(* IEC 61131-3 sources: elnaProjects/ElpcLogic/PomarKc7Unchanged/build_USO_ecl (part 5) *)

  resetDiProtection(protections.OsevojSdvigPravyjDi);
  resetDiProtection(protections.OsevojSdvigLevyjDi);
  resetDiProtection(protections.dP_masloGaz_LowDI);
  resetDiProtection(protections.DavlenieMaslaSmazkiDi);
  resetDiProtection(protections.mvOff);
  resetDiProtection(protections.NeispravnostVozbuzhdenijaDi);
  resetDiProtection(protections.AO_KC);
  resetDiProtection(protections.AO_PRU);
  resetDiProtection(protections.AO_SHU);
  resetDiProtection(protections.Srab_BEAO);
  resetDiProtection(protections.EAO_PRU);
  resetDiProtection(protections.BEAO_knSHU);
  resetDiProtection(protections.Kran1sdvig);
  resetDiProtection(protections.Kran2sdvig);
END_FUNCTION

FUNCTION BlockAllIM : BOOL
  VAR_IN_OUT
    IM : ImConfig;
  END_VAR

  IF NOT IM.Kran1.inOpcCommandsDisabled   THEN IM.Kran1.inOpcCommandsDisabled:=TRUE; END_IF;
  IF NOT IM.Kran2.inOpcCommandsDisabled   THEN IM.Kran2.inOpcCommandsDisabled:=TRUE; END_IF;
  IF NOT IM.Kran3b.inOpcCommandsDisabled  THEN IM.Kran3b.inOpcCommandsDisabled:=TRUE; END_IF;
  IF NOT IM.Kran4.inOpcCommandsDisabled   THEN IM.Kran4.inOpcCommandsDisabled:=TRUE; END_IF;
  IF NOT IM.Kran5.inOpcCommandsDisabled   THEN IM.Kran5.inOpcCommandsDisabled:=TRUE; END_IF;
  (*IF NOT IM.Kran6.inOpcCommandsDisabled   THEN IM.Kran6.inOpcCommandsDisabled:=TRUE; END_IF;*)

  IF NOT IM.nu1.inOpcCommandsDisabled     THEN IM.nu1.inOpcCommandsDisabled:=TRUE; END_IF;
  IF NOT IM.nu2.inOpcCommandsDisabled     THEN IM.nu2.inOpcCommandsDisabled:=TRUE; END_IF;
  IF NOT IM.pns.inOpcCommandsDisabled     THEN IM.pns.inOpcCommandsDisabled:=TRUE; END_IF;
  IF NOT IM.v1_Avom.inOpcCommandsDisabled THEN IM.v1_Avom.inOpcCommandsDisabled:=TRUE; END_IF;
  IF NOT IM.v2_Avom.inOpcCommandsDisabled THEN IM.v2_Avom.inOpcCommandsDisabled:=TRUE; END_IF;
  IF NOT IM.Ten.inOpcCommandsDisabled     THEN IM.Ten.inOpcCommandsDisabled:=TRUE; END_IF;
  IF NOT IM.mv.inOpcCommandsDisabled      THEN IM.mv.inOpcCommandsDisabled:=TRUE; END_IF;
END_FUNCTION

FUNCTION UnBlockAllIM : BOOL
  VAR_IN_OUT
    IM : ImConfig;
  END_VAR

  IF IM.TypeSwitch.Value = 1 THEN

  IF IM.Kran1.inOpcCommandsDisabled   THEN IM.Kran1.inOpcCommandsDisabled:=FALSE; END_IF;
  IF IM.Kran2.inOpcCommandsDisabled   THEN IM.Kran2.inOpcCommandsDisabled:=FALSE; END_IF;
  IF IM.Kran3b.inOpcCommandsDisabled  THEN IM.Kran3b.inOpcCommandsDisabled:=FALSE; END_IF;
  IF IM.Kran4.inOpcCommandsDisabled   THEN IM.Kran4.inOpcCommandsDisabled:=FALSE; END_IF;
  IF IM.Kran5.inOpcCommandsDisabled   THEN IM.Kran5.inOpcCommandsDisabled:=FALSE; END_IF;
  (*IF IM.Kran6.inOpcCommandsDisabled   THEN IM.Kran6.inOpcCommandsDisabled:=FALSE; END_IF;*)
  END_IF;

  IF IM.nu1.inOpcCommandsDisabled     THEN IM.nu1.inOpcCommandsDisabled:=FALSE; END_IF;
  IF IM.nu2.inOpcCommandsDisabled     THEN IM.nu2.inOpcCommandsDisabled:=FALSE; END_IF;
  IF IM.pns.inOpcCommandsDisabled     THEN IM.pns.inOpcCommandsDisabled:=FALSE; END_IF;
  IF IM.v1_Avom.inOpcCommandsDisabled THEN IM.v1_Avom.inOpcCommandsDisabled:=FALSE; END_IF;
  IF IM.v2_Avom.inOpcCommandsDisabled THEN IM.v2_Avom.inOpcCommandsDisabled:=FALSE; END_IF;
  IF IM.Ten.inOpcCommandsDisabled     THEN IM.Ten.inOpcCommandsDisabled:=FALSE; END_IF;
  IF IM.mv.inOpcCommandsDisabled      THEN IM.mv.inOpcCommandsDisabled:=FALSE; END_IF;
END_FUNCTION

FUNCTION_BLOCK RemontAlg
  VAR_IN_OUT
    StrAlg : struct_Alg;
  END_VAR
  VAR
    _sunpackerCommand : fb_sunpackerCommand;
    source : BYTE;
    cmd : BYTE;
    lastCmd : BYTE;
    source_for_Status : BYTE;
    cmd_for_Status : BYTE;
    command_error_for_Status : BYTE;
    resetCmdTimer : TON;
    resetCmdTimerPriznak : BOOL;
  END_VAR
  VAR_EXTERNAL
    protectManager : struct_ProtectionsManager;
    algManager : struct_AlgoritmsManager;
    ModeGpa : TYPE_ModeGpa;
    PMcommand : TYPE_CommandsPotectionsManager;
    IM : ImConfig;
  END_VAR

  StrAlg.CanRun := StrAlg.inCanRun;
  StrAlg.OpcCommandsDisabled := StrAlg.inOpcCommandsDisabled;

  (* ---- Если управление с ВУ заблокировано, то передаем команду из алгоритма ---- *)
  IF StrAlg.inOpcCommandsDisabled THEN
  	StrAlg.inCommand := StrAlg.inCommand_Alg;
  ELSE (* иначе передаем команду с АРМа*)
  	StrAlg.inCommand := StrAlg.inCommand_ARM;
  END_IF;

  _sunpackerCommand(command := StrAlg.inCommand);
  	source := _sunpackerCommand.source;
  	cmd := _sunpackerCommand.cmd;

  IF cmd <> 0 AND lastCmd <> cmd AND (((NOT StrAlg.opcCommandsDisabled) AND source > 0) OR source = 0) then
  	CASE BYTE_TO_INT(cmd) OF
  		(*cmdRun*) 1: 	IF (StrAlg.CanRun) THEN
  					StrAlg.isRuning := TRUE;
  					StrAlg.isEnded := FALSE;
  					StrAlg.hasError 	:= FALSE;
                                               (*****************       OnRun       *****************)
                                                        algManager.nMode:=ModeGpa.MODE_REMONT;
                                                        protectManager.inCommand:=PMcommand.ResetAllProtections;
  					    UnBlockAllIM(IM);
                                                    (*StrAlg.inOpcCommandsDisabled:=FALSE;*)
  					cmd_for_Status := cmd;
  					source_for_Status := source;
  					command_error_for_Status := 0;
  				ELSE
  					StrAlg.isRuning := FALSE;
  					StrAlg.isEnded := FALSE;
  					StrAlg.hasError 	:= FALSE;

  					cmd_for_Status := 0;
  					source_for_Status := source;
  					command_error_for_Status := cmd;
  				END_IF;
  		(*cmdReset*) 2: 	StrAlg.isRuning := FALSE;
  				StrAlg.isEnded := FALSE;
  				StrAlg.hasError 	:= FALSE;
                                          (*****************       OnReset       *****************)
                                                    BlockAllIM(IM);
                                                    protectManager.inCommand:=PMcommand.RestartAllProtections;
                                                    algManager.nMode:=ModeGpa.MODE_STOP;

  				cmd_for_Status := cmd;
  				source_for_Status := source;
  				command_error_for_Status := 0;
  	END_CASE;
  	resetCmdTimer(IN := false);
  	resetCmdTimerPriznak := TRUE;
  END_IF;
  lastCmd := cmd;

  resetCmdTimer(IN := resetCmdTimerPriznak, PT := T#5S);
  IF resetCmdTimer.Q THEN
  	resetCmdTimerPriznak := FALSE;
  	source_for_Status := 0;
  	cmd_for_Status := 0;
  	command_error_for_Status := 0;
  END_IF;

  StrAlg.status :=  SHL(BYTE_TO_DWORD(source_for_Status), 29)
  			OR SHL(BYTE_TO_DWORD(cmd_for_Status), 26)
  			OR SHL(BYTE_TO_DWORD(command_error_for_Status), 23)
  			OR SHL(BOOL_TO_DWORD(StrAlg.OpcCommandsDisabled ), 21)
  			OR SHL(BOOL_TO_DWORD(StrAlg.hasError),4)
  			OR SHL(BOOL_TO_DWORD(StrAlg.CanRun),2)
  			OR SHL(BOOL_TO_DWORD(StrAlg.isEnded),1)
  			OR BOOL_TO_DWORD(StrAlg.isRuning);
END_FUNCTION_BLOCK

FUNCTION EnableAiLimits : BOOL
  VAR_IN_OUT
    ai : AiConfig;
  END_VAR

  ai.P_masla_smazki_nizkoe.Disabled_LA:=FALSE;
   ai.P_masla_smazki_nizkoe.Disabled_LW:=FALSE;
   ai.P_masla_smazki_srednee_posle_nasosov.Disabled_LW:=FALSE;
   ai.dPmaslo_gaz.Disabled_LA:=FALSE;
   ai.dPmaslo_gaz.Disabled_LW:=FALSE;
END_FUNCTION

FUNCTION DisableAiLimits : BOOL
  VAR_IN_OUT
    ai : AiConfig;
  END_VAR

  ai.P_masla_smazki_nizkoe.Disabled_LA:=TRUE;
   ai.P_masla_smazki_nizkoe.Disabled_LW:=TRUE;
   ai.P_masla_smazki_srednee_posle_nasosov.Disabled_LW:=TRUE;
   ai.dPmaslo_gaz.Disabled_LA:=TRUE;
   ai.dPmaslo_gaz.Disabled_LW:=TRUE;
END_FUNCTION

FUNCTION_BLOCK TestProtectionAlg
  VAR_IN_OUT
    StrAlg : struct_Alg;
  END_VAR
  VAR
    _sunpackerCommand : fb_sunpackerCommand;
    source : BYTE;
    cmd : BYTE;
    lastCmd : BYTE;
    source_for_Status : BYTE;
    cmd_for_Status : BYTE;
    command_error_for_Status : BYTE;
    resetCmdTimer : TON;
    resetCmdTimerPriznak : BOOL;
  END_VAR
  VAR_EXTERNAL
    ai : AiConfig;
    protectManager : struct_ProtectionsManager;
    algManager : struct_AlgoritmsManager;
    ModeGpa : TYPE_ModeGpa;
    PMcommand : TYPE_CommandsPotectionsManager;
    IM : ImConfig;
  END_VAR

  StrAlg.CanRun := StrAlg.inCanRun;
  StrAlg.OpcCommandsDisabled := StrAlg.inOpcCommandsDisabled;

  (* ---- Если управление с ВУ заблокировано, то передаем команду из алгоритма ---- *)
  IF StrAlg.inOpcCommandsDisabled THEN
  	StrAlg.inCommand := StrAlg.inCommand_Alg;
  ELSE (* иначе передаем команду с АРМа*)
  	StrAlg.inCommand := StrAlg.inCommand_ARM;
  END_IF;

  _sunpackerCommand(command := StrAlg.inCommand);
  	source := _sunpackerCommand.source;
  	cmd := _sunpackerCommand.cmd;

  IF cmd <> 0 AND lastCmd <> cmd AND (((NOT StrAlg.opcCommandsDisabled) AND source > 0) OR source = 0) then
  	CASE BYTE_TO_INT(cmd) OF
  		(*cmdRun*) 1: 	IF (StrAlg.CanRun) THEN
  					StrAlg.isRuning := TRUE;
  					StrAlg.isEnded := FALSE;
  					StrAlg.hasError 	:= FALSE;
                                               (*****************       OnRun       *****************)
                                                        algManager.nMode:=ModeGpa.MODE_TESTAZ;
                                                        protectManager.inCommand:=PMcommand.CheckProtections;
  					    EnableAiLimits(ai);
                                                        IM.SingleSignals.P_oil_low.Disabled_Sig:=FALSE;
                                                        IM.SingleSignals.dP_oilgaz_low.Disabled_Sig:=FALSE;
                                                    (*StrAlg.inOpcCommandsDisabled:=FALSE;*)
  					cmd_for_Status := cmd;
  					source_for_Status := source;
  					command_error_for_Status := 0;
  				ELSE
  					StrAlg.isRuning := FALSE;
  					StrAlg.isEnded := FALSE;
  					StrAlg.hasError 	:= FALSE;

  					cmd_for_Status := 0;
  					source_for_Status := source;
  					command_error_for_Status := cmd;
  				END_IF;
  		(*cmdReset*) 2: 	StrAlg.isRuning := FALSE;
  				StrAlg.isEnded := FALSE;
  				StrAlg.hasError 	:= FALSE;
                                          (*****************       OnReset       *****************)
                                                    DisableAiLimits(ai);
                                                    IM.SingleSignals.P_oil_low.Disabled_Sig:=TRUE;
                                                    IM.SingleSignals.dP_oilgaz_low.Disabled_Sig:=TRUE;
                                                    protectManager.inCommand:=PMcommand.RestartAllProtections;
                                                    algManager.nMode:=ModeGpa.MODE_STOP;

  				cmd_for_Status := cmd;
  				source_for_Status := source;
  				command_error_for_Status := 0;
  	END_CASE;
  	resetCmdTimer(IN := false);
  	resetCmdTimerPriznak := TRUE;
  END_IF;
  lastCmd := cmd;

  resetCmdTimer(IN := resetCmdTimerPriznak, PT := T#5S);
  IF resetCmdTimer.Q THEN
  	resetCmdTimerPriznak := FALSE;
  	source_for_Status := 0;
  	cmd_for_Status := 0;
  	command_error_for_Status := 0;
  END_IF;

  StrAlg.status :=  SHL(BYTE_TO_DWORD(source_for_Status), 29)
  			OR SHL(BYTE_TO_DWORD(cmd_for_Status), 26)
  			OR SHL(BYTE_TO_DWORD(command_error_for_Status), 23)
  			OR SHL(BOOL_TO_DWORD(StrAlg.OpcCommandsDisabled ), 21)
  			OR SHL(BOOL_TO_DWORD(StrAlg.hasError),4)
  			OR SHL(BOOL_TO_DWORD(StrAlg.CanRun),2)
  			OR SHL(BOOL_TO_DWORD(StrAlg.isEnded),1)
  			OR BOOL_TO_DWORD(StrAlg.isRuning);
END_FUNCTION_BLOCK

FUNCTION_BLOCK TestImAlg
  VAR_IN_OUT
    StrAlg : struct_Alg;
  END_VAR
  VAR
    _sunpackerCommand : fb_sunpackerCommand;
    source : BYTE;
    cmd : BYTE;
    lastCmd : BYTE;
    source_for_Status : BYTE;
    cmd_for_Status : BYTE;
    command_error_for_Status : BYTE;
    resetCmdTimer : TON;
    resetCmdTimerPriznak : BOOL;
  END_VAR
  VAR_EXTERNAL
    protectManager : struct_ProtectionsManager;
    algManager : struct_AlgoritmsManager;
    ModeGpa : TYPE_ModeGpa;
    PMcommand : TYPE_CommandsPotectionsManager;
    IM : ImConfig;
  END_VAR

  StrAlg.CanRun := StrAlg.inCanRun;
  StrAlg.OpcCommandsDisabled := StrAlg.inOpcCommandsDisabled;

  (* ---- Если управление с ВУ заблокировано, то передаем команду из алгоритма ---- *)
  IF StrAlg.inOpcCommandsDisabled THEN
  	StrAlg.inCommand := StrAlg.inCommand_Alg;
  ELSE (* иначе передаем команду с АРМа*)
  	StrAlg.inCommand := StrAlg.inCommand_ARM;
  END_IF;

  _sunpackerCommand(command := StrAlg.inCommand);
  	source := _sunpackerCommand.source;
  	cmd := _sunpackerCommand.cmd;

  IF cmd <> 0 AND lastCmd <> cmd AND (((NOT StrAlg.opcCommandsDisabled) AND source > 0) OR source = 0) then
  	CASE BYTE_TO_INT(cmd) OF
  		(*cmdRun*) 1: 	IF (StrAlg.CanRun) THEN
  					StrAlg.isRuning := TRUE;
  					StrAlg.isEnded := FALSE;
  					StrAlg.hasError 	:= FALSE;
                                               (*****************       OnRun       *****************)

                                                        algManager.nMode:=ModeGpa.MODE_TESTIM;
  					    UnBlockAllIM(IM);

                                                    (*StrAlg.inOpcCommandsDisabled:=FALSE;*)
  					cmd_for_Status := cmd;
  					source_for_Status := source;
  					command_error_for_Status := 0;
  				ELSE
  					StrAlg.isRuning := FALSE;
  					StrAlg.isEnded := FALSE;
  					StrAlg.hasError 	:= FALSE;

  					cmd_for_Status := 0;
  					source_for_Status := source;
  					command_error_for_Status := cmd;
  				END_IF;
  		(*cmdReset*) 2: 	StrAlg.isRuning := FALSE;
  				StrAlg.isEnded := FALSE;
  				StrAlg.hasError 	:= FALSE;
                                          (*****************       OnReset       *****************)
                                                    BlockAllIM(IM);
                                                    algManager.nMode:=ModeGpa.MODE_STOP;

  				cmd_for_Status := cmd;
  				source_for_Status := source;
  				command_error_for_Status := 0;
  	END_CASE;
  	resetCmdTimer(IN := false);
  	resetCmdTimerPriznak := TRUE;
  END_IF;
  lastCmd := cmd;

  resetCmdTimer(IN := resetCmdTimerPriznak, PT := T#5S);
  IF resetCmdTimer.Q THEN
  	resetCmdTimerPriznak := FALSE;
  	source_for_Status := 0;
  	cmd_for_Status := 0;
  	command_error_for_Status := 0;
  END_IF;

  StrAlg.status :=  SHL(BYTE_TO_DWORD(source_for_Status), 29)
  			OR SHL(BYTE_TO_DWORD(cmd_for_Status), 26)
  			OR SHL(BYTE_TO_DWORD(command_error_for_Status), 23)
  			OR SHL(BOOL_TO_DWORD(StrAlg.OpcCommandsDisabled ), 21)
  			OR SHL(BOOL_TO_DWORD(StrAlg.hasError),4)
  			OR SHL(BOOL_TO_DWORD(StrAlg.CanRun),2)
  			OR SHL(BOOL_TO_DWORD(StrAlg.isEnded),1)
  			OR BOOL_TO_DWORD(StrAlg.isRuning);
END_FUNCTION_BLOCK

FUNCTION_BLOCK fb_AutoTenAlg
  VAR_IN_OUT
    StrAlg : struct_Alg;
    PNS : struct_Switch;
    TEN : struct_Switch;
  END_VAR
  VAR_INPUT
    T_masla : struct_AI;
    Uroven_masla : struct_AI;
    offTemperature : struct_AnalogParametr;
  END_VAR
  VAR
    _sunpackerCommand : fb_sunpackerCommand;
    _statusAi : TYPE_StatusAi;
    _statusDualInput : TYPE_statusDualInput;
    _commandDualInput : TYPE_commandDualInput;
    source : BYTE;
    cmd : BYTE;
    lastCmd : BYTE;
    source_for_Status : BYTE;
    cmd_for_Status : BYTE;
    command_error_for_Status : BYTE;
    resetCmdTimer : TON;
    resetCmdTimerPriznak : BOOL;
    onInit : BOOL;
  END_VAR

  IF NOT onInit THEN
  StrAlg.inCanRun:=TRUE;
  onInit:=TRUE;
  END_IF;

  IF StrAlg.isRuning THEN

  IF ((T_masla.interval >= _statusAi.normal) AND (T_masla.value > offTemperature.Value)) OR
  ((Uroven_masla.interval >= _statusAi.normal) AND (Uroven_masla.value < Uroven_masla.LA)) OR
  (PNS.onStatus=_statusDualInput.STATUS_OFF) THEN

        TEN.inOpcCommandsDisabled:=TRUE;

  	IF TEN.onStatus = _statusDualInput.STATUS_ON THEN
            TEN.inCommand_Alg:=BYTE_TO_WORD(_commandDualInput.CMD_OFF);
  	END_IF;

  ELSIF PNS.onStatus = _statusDualInput.STATUS_ON THEN
        TEN.inOpcCommandsDisabled:=FALSE;
  END_IF;

  END_IF;

  StrAlg.CanRun := StrAlg.inCanRun;
  StrAlg.hasError := TEN.CommandFault OR (T_masla.interval < _statusAi.normal) OR (Uroven_masla.interval < _statusAi.normal);

  StrAlg.OpcCommandsDisabled := StrAlg.inOpcCommandsDisabled;

  (* ---- Если управление с ВУ заблокировано, то  передаем команду из алгоритма ---- *)
  IF StrAlg.inOpcCommandsDisabled THEN
  	StrAlg.inCommand := StrAlg.inCommand_Alg;
  ELSE (* иначе передаем команду с АРМа*)
  	StrAlg.inCommand := StrAlg.inCommand_ARM;
  END_IF;

  _sunpackerCommand(command := StrAlg.inCommand);
  	source := _sunpackerCommand.source;
  	cmd := _sunpackerCommand.cmd;

  IF cmd <> 0 AND lastCmd <> cmd AND (((NOT StrAlg.opcCommandsDisabled) AND source > 0) OR source = 0) then
  	CASE BYTE_TO_INT(cmd) OF
  		(*cmdRun*) 1: 	IF StrAlg.CanRun AND NOT StrAlg.hasError THEN
  					StrAlg.isRuning := TRUE;
  					StrAlg.isEnded := FALSE;
  					(*StrAlg.hasError := FALSE;*)

                                                    (*****************       OnRun       *****************)
                                                    IF StrAlg.inOpcCommandsDisabled THEN
  		                              StrAlg.inOpcCommandsDisabled:=FALSE;
                                                    END_IF;
  					cmd_for_Status := cmd;
  					source_for_Status := source;
  					command_error_for_Status := 0;
  				ELSE
  					StrAlg.isRuning := FALSE;
  					StrAlg.isEnded := FALSE;
  					(*StrAlg.hasError 	:= FALSE;*)

  					cmd_for_Status := 0;
  					source_for_Status := source;
  					command_error_for_Status := cmd;
  				END_IF;
  		(*cmdReset*) 2: 	StrAlg.isRuning := FALSE;
  				StrAlg.isEnded := FALSE;
  				(*StrAlg.hasError 	:= FALSE;*)

                                          (*****************       OnReset       *****************)
                                          TEN.inOpcCommandsDisabled:=TRUE;
                                          TEN.inCommand_Alg:=BYTE_TO_WORD(_commandDualInput.CMD_OFF);

  				cmd_for_Status := cmd;
  				source_for_Status := source;
  				command_error_for_Status := 0;
  	END_CASE;
  	resetCmdTimer(IN := false);
  	resetCmdTimerPriznak := TRUE;
  END_IF;
  lastCmd := cmd;

  resetCmdTimer(IN := resetCmdTimerPriznak, PT := T#5S);
  IF resetCmdTimer.Q THEN
  	resetCmdTimerPriznak := FALSE;
  	source_for_Status := 0;
  	cmd_for_Status := 0;
  	command_error_for_Status := 0;
  END_IF;

  (*TODO: TYPE PROGRAM CODE HERE*)
  StrAlg.status :=  SHL(BYTE_TO_DWORD(source_for_Status), 29)
  			OR SHL(BYTE_TO_DWORD(cmd_for_Status), 26)
  			OR SHL(BYTE_TO_DWORD(command_error_for_Status), 23)
  			OR SHL(BOOL_TO_DWORD(StrAlg.OpcCommandsDisabled ), 21)
  			OR SHL(BOOL_TO_DWORD(StrAlg.hasError),4)
  			OR SHL(BOOL_TO_DWORD(StrAlg.CanRun),2)
  			OR SHL(BOOL_TO_DWORD(StrAlg.isEnded),1)
  			OR BOOL_TO_DWORD(StrAlg.isRuning);
END_FUNCTION_BLOCK

FUNCTION_BLOCK fb_AutoPnsAlg
  VAR_IN_OUT
    StrAlg : struct_Alg;
    Nasos : struct_Switch;
  END_VAR
  VAR_INPUT
    diPlow : struct_singleSignal;
    Poil : struct_AI;
    Ust_Run : struct_AnalogParametr;
    Ust_Stop : struct_AnalogParametr;
  END_VAR
  VAR
    _sunpackerCommand : fb_sunpackerCommand;
    _statusAi : TYPE_StatusAi;
    _statusDualInput : TYPE_statusDualInput;
    _commandDualInput : TYPE_commandDualInput;
    source : BYTE;
    cmd : BYTE;
    lastCmd : BYTE;
    source_for_Status : BYTE;
    cmd_for_Status : BYTE;
    command_error_for_Status : BYTE;
    resetCmdTimer : TON;
    resetCmdTimerPriznak : BOOL;
    onInit : BOOL;
    onTrig : R_TRIG;
    offTrig : R_TRIG;
    waitOn : TON;
    waitOff : TON;
  END_VAR
  VAR_EXTERNAL
    AlgTimers : struct_AlgTimers;
  END_VAR

  IF NOT onInit THEN
  StrAlg.inOpcCommandsDisabled:=TRUE;
  StrAlg.inCanRun:=TRUE;
  onInit:=TRUE;
  END_IF;

  IF StrAlg.isRuning THEN

  StrAlg.hasError := Nasos.CommandFault OR (Poil.interval < _statusAi.normal OR NOT diPlow.reliability);

      IF (Poil.Interval >= _statusAi.normal) THEN
      waitOn(IN:=Poil.Value <= Ust_Run.value OR diPlow.q, PT := T#1S);
      waitOff(IN:= Poil.Value >= Ust_Stop.value, PT := T#300S);

      ELSE
      waitOn(IN:=diPlow.Q, PT := T#1S);
      END_IF;

  onTrig(CLK:=waitOn.Q);
  offTrig(CLK:=waitOff.Q);
      IF (Poil.Value>=Ust_Stop.value) AND Nasos.inopcCommandsDisabled THEN
          Nasos.inopcCommandsDisabled:=FALSE;
      END_IF;

      IF onTrig.Q THEN
      Nasos.inopcCommandsDisabled:=TRUE;
      Nasos.inCommand_Alg:=BYTE_TO_WORD(_commandDualInput.CMD_ON);
      END_IF;

      IF offTrig.Q THEN
          IF NOT (Nasos.onStatus=_statusDualInput.STATUS_OFF) THEN
          Nasos.inopcCommandsDisabled:=TRUE;
          Nasos.inCommand_Alg:=BYTE_TO_WORD(_commandDualInput.CMD_OFF);
          END_IF;
      END_IF;

  AlgTimers.AutoPns_OnTimer:=UDINT_TO_UINT(TIME_TO_UDINT(waitOn.PT - waitOn.ET)/1000);
  AlgTimers.AutoPns_OffTimer:=UDINT_TO_UINT(TIME_TO_UDINT(waitOff.PT -waitOff.ET)/1000);

  END_IF;

  StrAlg.CanRun := StrAlg.inCanRun;

  StrAlg.OpcCommandsDisabled := StrAlg.inOpcCommandsDisabled;

  (* ---- Если управление с ВУ заблокировано, то  передаем команду из алгоритма ---- *)
  IF StrAlg.inOpcCommandsDisabled THEN
  	StrAlg.inCommand := StrAlg.inCommand_Alg;
  ELSE (* иначе передаем команду с АРМа*)
  	StrAlg.inCommand := StrAlg.inCommand_ARM;
  END_IF;

  _sunpackerCommand(command := StrAlg.inCommand);
  	source := _sunpackerCommand.source;
  	cmd := _sunpackerCommand.cmd;

  IF cmd <> 0 AND lastCmd <> cmd AND (((NOT StrAlg.opcCommandsDisabled) AND source > 0) OR source = 0) then
  	CASE BYTE_TO_INT(cmd) OF
  		(*cmdRun*) 1: 	IF (StrAlg.CanRun) THEN
  					StrAlg.isRuning := TRUE;
  					StrAlg.isEnded := FALSE;
  					StrAlg.hasError := FALSE;
  					(*****************       OnRun       *****************)

  					cmd_for_Status := cmd;
  					source_for_Status := source;
  					command_error_for_Status := 0;
  				ELSE
  					StrAlg.isRuning := FALSE;
  					StrAlg.isEnded := FALSE;
  					StrAlg.hasError 	:= FALSE;

  					cmd_for_Status := 0;
  					source_for_Status := source;
  					command_error_for_Status := cmd;
  				END_IF;
  		(*cmdReset*) 2: 	StrAlg.isRuning := FALSE;
  				StrAlg.isEnded := FALSE;
  				StrAlg.hasError 	:= FALSE;

                                           (*****************       OnReset       *****************)
                                          waitOn(in:=FALSE);
                                          waitOff(in:=FALSE);
                                          AlgTimers.AutoPns_OffTimer:=UDINT_TO_UINT(TIME_TO_UDINT(waitOff.pt -waitOff.ET)/1000);

  				cmd_for_Status := cmd;
  				source_for_Status := source;
  				command_error_for_Status := 0;
  	END_CASE;
  	resetCmdTimer(IN := false);
  	resetCmdTimerPriznak := TRUE;
  END_IF;
  lastCmd := cmd;

  resetCmdTimer(IN := resetCmdTimerPriznak, PT := T#5S);
  IF resetCmdTimer.Q THEN
  	resetCmdTimerPriznak := FALSE;
  	source_for_Status := 0;
  	cmd_for_Status := 0;
  	command_error_for_Status := 0;
  END_IF;

  (*TODO: TYPE PROGRAM CODE HERE*)
  StrAlg.status :=  SHL(BYTE_TO_DWORD(source_for_Status), 29)
  			OR SHL(BYTE_TO_DWORD(cmd_for_Status), 26)
  			OR SHL(BYTE_TO_DWORD(command_error_for_Status), 23)
  			OR SHL(BOOL_TO_DWORD(StrAlg.OpcCommandsDisabled ), 21)
  			OR SHL(BOOL_TO_DWORD(StrAlg.hasError),4)
  			OR SHL(BOOL_TO_DWORD(StrAlg.CanRun),2)
  			OR SHL(BOOL_TO_DWORD(StrAlg.isEnded),1)
  			OR BOOL_TO_DWORD(StrAlg.isRuning);
END_FUNCTION_BLOCK

FUNCTION_BLOCK fb_AutoAvomAlg
  VAR_IN_OUT
    StrAlg : struct_Alg;
    im1 : struct_Switch;
    im2 : struct_Switch;
  END_VAR
  VAR_INPUT
    ai : struct_AI;
  END_VAR
  VAR_IN_OUT
    on1Temperature : struct_AnalogParametr;
    on2Temperature : struct_AnalogParametr;
    hystereses : struct_AnalogParametr;
  END_VAR
  VAR
    _sunpackerCommand : fb_sunpackerCommand;
    _statusAi : TYPE_StatusAi;
    _statusDualInput : TYPE_statusDualInput;
    _commandDualInput : TYPE_commandDualInput;
    source : BYTE;
    cmd : BYTE;
    lastCmd : BYTE;
    source_for_Status : BYTE;
    cmd_for_Status : BYTE;
    command_error_for_Status : BYTE;
    resetCmdTimer : TON;
    resetCmdTimerPriznak : BOOL;
    onInit : BOOL;
  END_VAR

  (*
  IF NOT onInit THEN
  StrAlg.inCanRun:=TRUE;
  onInit:=TRUE;
  END_IF;
  *)

  IF StrAlg.isRuning THEN

  StrAlg.hasError := im1.CommandFault OR im2.CommandFault OR (ai.interval<_statusAi.normal);

      IF (ai.interval>=_statusAi.normal) THEN

            IF (ai.value>= on1Temperature.Value) THEN
                IF im1.onStatus <> _statusDualInput.STATUS_ON THEN
  	       im1.inCommand_Alg:=BYTE_TO_WORD(_commandDualInput.CMD_ON); (*cmd_on*)
                END_IF;
            END_IF;

            IF  ai.value < (on1Temperature.Value - hystereses.Value) THEN
                IF im1.onStatus <> _statusDualInput.STATUS_OFF THEN
  	       im1.inCommand_Alg:=BYTE_TO_WORD(_commandDualInput.CMD_OFF);
                END_IF;
            END_IF;

             IF (ai.value>= on2Temperature.Value) THEN
                IF im2.onStatus <> _statusDualInput.STATUS_ON THEN
  	       im2.inCommand_Alg:=BYTE_TO_WORD(_commandDualInput.CMD_ON); (*cmd_on*)
                END_IF;
            END_IF;

            IF  ai.value < (on2Temperature.Value - hystereses.Value) THEN
                IF im2.onStatus <> _statusDualInput.STATUS_OFF THEN
  	       im2.inCommand_Alg:=BYTE_TO_WORD(_commandDualInput.CMD_OFF);
                END_IF;
            END_IF;
       END_IF;

  END_IF;

  StrAlg.CanRun := StrAlg.inCanRun;

  StrAlg.OpcCommandsDisabled := StrAlg.inOpcCommandsDisabled;

  (* ---- Если управление с ВУ заблокировано, то  передаем команду из алгоритма ---- *)
  IF StrAlg.inOpcCommandsDisabled THEN
  	StrAlg.inCommand := StrAlg.inCommand_Alg;
  ELSE (* иначе передаем команду с АРМа*)
  	StrAlg.inCommand := StrAlg.inCommand_ARM;
  END_IF;

  _sunpackerCommand(command := StrAlg.inCommand);
  	source := _sunpackerCommand.source;
  	cmd := _sunpackerCommand.cmd;

  IF cmd <> 0 AND lastCmd <> cmd AND (((NOT StrAlg.opcCommandsDisabled) AND source > 0) OR source = 0) then
  	CASE BYTE_TO_INT(cmd) OF
  		(*cmdRun*) 1: 	IF (StrAlg.CanRun) THEN
  					StrAlg.isRuning := TRUE;
  					StrAlg.isEnded := FALSE;
  					StrAlg.hasError := FALSE;
                                                    StrAlg.inOpcCommandsDisabled:=FALSE;
  					im1.inOpcCommandsDisabled:=TRUE;
                                                    im2.inOpcCommandsDisabled:=TRUE;
  					cmd_for_Status := cmd;
  					source_for_Status := source;
  					command_error_for_Status := 0;
  				ELSE
  					StrAlg.isRuning := FALSE;
  					StrAlg.isEnded := FALSE;
  					StrAlg.hasError 	:= FALSE;

  					cmd_for_Status := 0;
  					source_for_Status := source;
  					command_error_for_Status := cmd;
  				END_IF;
  		(*cmdReset*) 2: 	StrAlg.isRuning := FALSE;
  				StrAlg.isEnded := FALSE;
  				StrAlg.hasError 	:= FALSE;
                                          StrAlg.inOpcCommandsDisabled:=FALSE;
                                          im1.inOpcCommandsDisabled:=FALSE;
                                          im2.inOpcCommandsDisabled:=FALSE;
                                          im1.inCommand_Alg:=0;
                                          im2.inCommand_Alg:=0;
  				cmd_for_Status := cmd;
  				source_for_Status := source;
  				command_error_for_Status := 0;
  	END_CASE;
  	resetCmdTimer(IN := false);
  	resetCmdTimerPriznak := TRUE;
  END_IF;
  lastCmd := cmd;

  resetCmdTimer(IN := resetCmdTimerPriznak, PT := T#5S);
  IF resetCmdTimer.Q THEN
  	resetCmdTimerPriznak := FALSE;
  	source_for_Status := 0;
  	cmd_for_Status := 0;
  	command_error_for_Status := 0;
  END_IF;

  (*TODO: TYPE PROGRAM CODE HERE*)
  StrAlg.status :=  SHL(BYTE_TO_DWORD(source_for_Status), 29)
  			OR SHL(BYTE_TO_DWORD(cmd_for_Status), 26)
  			OR SHL(BYTE_TO_DWORD(command_error_for_Status), 23)
  			OR SHL(BOOL_TO_DWORD(StrAlg.OpcCommandsDisabled ), 21)
  			OR SHL(BOOL_TO_DWORD(StrAlg.hasError),4)
  			OR SHL(BOOL_TO_DWORD(StrAlg.CanRun),2)
  			OR SHL(BOOL_TO_DWORD(StrAlg.isEnded),1)
  			OR BOOL_TO_DWORD(StrAlg.isRuning);
END_FUNCTION_BLOCK

FUNCTION resetIfRunning : BOOL
  VAR_IN_OUT
    alg : struct_Alg;
  END_VAR
  VAR CONSTANT
    cmdReset : WORD := 2;
  END_VAR

  IF alg.isRuning THEN
                      alg.inOpcCommandsDisabled:=TRUE;
  		alg.inCommand_Alg:=cmdReset;
  END_IF;
END_FUNCTION

FUNCTION runIfNotRunning : BOOL
  VAR_IN_OUT
    alg : struct_Alg;
  END_VAR
  VAR CONSTANT
    cmdRun : WORD := 1;
  END_VAR

  IF NOT alg.isRuning THEN
                      alg.inOpcCommandsDisabled:=TRUE;
                      alg.inCanRun:=TRUE;
  		alg.inCommand_Alg:=cmdRun;
  END_IF;
END_FUNCTION

FUNCTION_BLOCK fb_ph_algoritm
  VAR_IN_OUT
    alg : struct_Alg;
  END_VAR
  VAR_INPUT
    act : TYPE_PhaseAlgoritmAction;
    PhaseNumber : UINT;
    waitCompletion : BOOL;
  END_VAR
  VAR_IN_OUT
    StrPh : struct_PhaseAlgoritm;
  END_VAR
  VAR
    CommandFault_Trig : R_TRIG;
    reset_Trig : R_TRIG;
    _statusDualInput : TYPE_statusDualInput;
  END_VAR

  IF StrPh.run AND NOT StrPh.start THEN
  	StrPh.start := TRUE;
  	StrPh.top := FALSE;
  	StrPh.error := FALSE;
            StrPh.run:=FALSE;

  	CASE act OF
  		(*PhaseAlgoritmAction.run*)    _run : runIfNotRunning(alg); (*cmd_run*)
  		(*PhaseAlgoritmAction.reset*)_reset : resetIfRunning(alg); (*cmd_reset*)
  	END_CASE;
  END_IF;

  IF StrPh.start AND NOT StrPh.top THEN
                      CommandFault_Trig(CLK := alg.hasError);
                      IF CommandFault_Trig.Q THEN
  	          StrPh.error := TRUE;
                      END_IF;

  		CASE act OF
  		(*PhaseAlgoritmAction.run*)    _run:
                                                          IF waitCompletion THEN
  		                                	StrPh.top:=alg.isEnded;
  		                                    ELSE
  			                              StrPh.top:=alg.isRuning;
  		                                    END_IF;

  		(*PhaseAlgoritmAction.reset*) _reset:   StrPh.top := NOT alg.isRuning;
  		END_CASE;

  END_IF;

  IF StrPh.top THEN
  StrPh.error := FALSE;
  END_IF;

  reset_Trig(CLK := StrPh.reset);
  IF reset_Trig.Q THEN
            IF waitCompletion THEN
            resetIfRunning(alg);
            END_IF;
  	StrPh.start := FALSE;
  	StrPh.error := FALSE;
  	StrPh.top := FALSE;
            StrPh.run:=FALSE;
            StrPh.reset:=FALSE;
  END_IF;

  StrPh.startStatus := SHL(BOOL_TO_DWORD(StrPh.start), PhaseNumber);
  StrPh.errorStatus := SHL(BOOL_TO_DWORD(StrPh.error), PhaseNumber);
  StrPh.topStatus := SHL(BOOL_TO_DWORD(StrPh.top), PhaseNumber);
END_FUNCTION_BLOCK

FUNCTION_BLOCK fb_ph_Timer
  VAR_INPUT
    delay : TIME;
    PhaseNumber : UINT;
  END_VAR
  VAR_IN_OUT
    StrPh : struct_PhaseAlgoritm;
  END_VAR
  VAR
    CommandFault_Trig : R_TRIG;
    reset_Trig : R_TRIG;
  END_VAR
  VAR_IN_OUT
    timer : UINT;
  END_VAR
  VAR
    _timer : TON;
    _statusDualInput : TYPE_statusDualInput;
  END_VAR

  IF StrPh.run AND NOT StrPh.start THEN
  	StrPh.start := TRUE;
  	StrPh.top := FALSE;
  	StrPh.error := FALSE;
            StrPh.run:=FALSE;

  END_IF;

  _timer(IN:=StrPh.start, PT:=delay);

  timer:=TIME_TO_UINT(delay -_timer.ET);

  IF StrPh.start AND NOT StrPh.top THEN
  StrPh.top:=_timer.Q;
  END_IF;

  reset_Trig(CLK := StrPh.reset);
  IF reset_Trig.Q THEN
  	StrPh.start := FALSE;
  	StrPh.error := FALSE;
  	StrPh.top := FALSE;
            StrPh.run:=FALSE;
            (*timer:=TIME_TO_UINT(delay -_timer.ET);*)
            StrPh.reset:=FALSE;
  END_IF;

  StrPh.startStatus := SHL(BOOL_TO_DWORD(StrPh.start), PhaseNumber);
  StrPh.errorStatus := SHL(BOOL_TO_DWORD(StrPh.error), PhaseNumber);
  StrPh.topStatus := SHL(BOOL_TO_DWORD(StrPh.top), PhaseNumber);
END_FUNCTION_BLOCK

FUNCTION_BLOCK fb_Question
  VAR_IN_OUT
    StrQ : struct_Question;
  END_VAR
  VAR
    Asked : UINT;
    _answers : TYPE_Answers;
  END_VAR
  VAR CONSTANT
    cmd_answer : UINT := 1;
  END_VAR
  VAR
    _sunpackerCommand : fb_sunpackerCommand;
    source : BYTE;
    parametr : BYTE;
    lastParametr : BYTE;
    cmd : BYTE;
    source_for_Status : BYTE;
    cmd_for_Status : BYTE;
    command_error_for_Status : BYTE;
    resetCmdTimer : TON;
    resetCmdTimerPriznak : BOOL;
    reset_Trig : R_TRIG;
  END_VAR

  StrQ.OpcCommandsDisabled := StrQ.inopcCommandsDisabled;

  IF StrQ.ask THEN
  StrQ.inopcCommandsDisabled:=FALSE;
      IF Asked=0 THEN
  	Asked:=StrQ.AnswerVariants;
  	StrQ.answer:=_answers.ANS_NONE;
      END_IF;

      _sunpackerCommand(command := StrQ.inCommand);
  	source := _sunpackerCommand.source;
            parametr := _sunpackerCommand.parametr;
  	cmd := _sunpackerCommand.cmd;

      IF cmd <> 0 AND lastParametr <> parametr AND ((NOT StrQ.OpcCommandsDisabled) AND source > 0)  then
  	CASE BYTE_TO_INT(cmd) OF
  	                               1 :

  				IF Asked<>0 THEN
                                             (* CASE BYTE_TO_INT(parametr) OF
                                              1: answer:=_answers.ANS_YES;
                                              2: answer:=_answers.ANS_NO;
                                              4: answer:=_answers.ANS_CANCEL;
                                              8: answer:=_answers.ANS_RETRY;
  	                                  END_CASE;*)
                                          StrQ.answer:=BYTE_TO_UINT(parametr);
                                          command_error_for_Status := 0;
                                          ELSE
  	                              command_error_for_Status := cmd;
                                          END_IF;
  	END_CASE;
  	source_for_Status := source;
  	cmd_for_Status := cmd;
  	resetCmdTimer(IN := FALSE);
  	resetCmdTimerPriznak := TRUE;
      END_IF;

      lastParametr := parametr;

      resetCmdTimer(IN := resetCmdTimerPriznak, PT := T#5S);
      IF resetCmdTimer.Q THEN
  	resetCmdTimerPriznak := FALSE;
  	source_for_Status := 0;
  	cmd_for_Status := 0;
  	command_error_for_Status := 0;
      END_IF;
  END_IF;

  reset_Trig(CLK := StrQ.reset);
  IF reset_Trig.Q THEN
  	Asked:=0;
  	StrQ.answer:=0;
            StrQ.ask:=FALSE;
            StrQ.reset:=FALSE;
  	StrQ.inopcCommandsDisabled:=TRUE;
  END_IF;

  StrQ.status := SHL(BYTE_TO_DWORD(source_for_Status), 29)
  			OR SHL(BYTE_TO_DWORD(cmd_for_Status), 26)
  			OR SHL(BYTE_TO_DWORD(command_error_for_Status), 23)
  			OR SHL(BOOL_TO_DWORD(StrQ.OpcCommandsDisabled ), 21);
  IF StrQ.answer = 0 THEN
      StrQ.status := StrQ.status  OR SHL(UINT_TO_DWORD(asked), 6);
  ELSE
      StrQ.status := StrQ.status  OR SHL(UINT_TO_DWORD(StrQ.answer), 6);
  END_IF;
END_FUNCTION_BLOCK

FUNCTION_BLOCK fb_ph_Switch
  VAR_IN_OUT
    im : struct_Switch;
  END_VAR
  VAR_INPUT
    act : TYPE_DualStateImAction;
    PhaseNumber : UINT;
  END_VAR
  VAR_IN_OUT
    StrPh : struct_PhaseAlgoritm;
  END_VAR
  VAR
    CommandFault_Trig : R_TRIG;
    reset_Trig : R_TRIG;
    _statusDualInput : TYPE_statusDualInput;
  END_VAR

  IF StrPh.run AND NOT StrPh.start THEN
  	StrPh.start := TRUE;
  	StrPh.top := FALSE;
  	StrPh.error := FALSE;
            StrPh.run:=FALSE;

  	CASE act OF
  		(*DualStateImAction.on*)   _on :im.inOpcCommandsDisabled:=TRUE;
                                                      im.inCommand_Alg := 1; (*cmd_open*)
  		(*DualStateImAction.off*) _off :im.inOpcCommandsDisabled:=TRUE;
                                                      im.inCommand_Alg := 2; (*cmd_close*)
  	END_CASE;
  END_IF;

  IF StrPh.start AND NOT StrPh.top THEN
                      CommandFault_Trig(CLK := im.CommandFault);
                      IF CommandFault_Trig.Q THEN
  	          StrPh.error := TRUE;
                      END_IF;

  		CASE act OF
  		(*_DualStateImAction.on*)    _on: StrPh.top := im.onStatus = _statusDualInput.STATUS_ON;
  		(*_DualStateImAction.off*)  _off: StrPh.top := im.onStatus = _statusDualInput.STATUS_OFF;
  		END_CASE;

  END_IF;

  IF StrPh.top THEN
  StrPh.error := FALSE;
  END_IF;

  reset_Trig(CLK := StrPh.reset);
  IF reset_Trig.Q THEN
  	StrPh.start := FALSE;
  	StrPh.error := FALSE;
  	StrPh.top := FALSE;
            StrPh.run:=FALSE;
            StrPh.reset:=FALSE;
  END_IF;

  StrPh.startStatus := SHL(BOOL_TO_DWORD(StrPh.start), PhaseNumber);
  StrPh.errorStatus := SHL(BOOL_TO_DWORD(StrPh.error), PhaseNumber);
  StrPh.topStatus := SHL(BOOL_TO_DWORD(StrPh.top), PhaseNumber);
END_FUNCTION_BLOCK

FUNCTION_BLOCK fb_ph_CustomPhase
  VAR_INPUT
    PhaseNumber : UINT;
  END_VAR
  VAR_IN_OUT
    StrPh : struct_PhaseAlgoritm;
  END_VAR
  VAR
    CommandFault_Trig : R_TRIG;
    reset_Trig : R_TRIG;
    _statusDualInput : TYPE_statusDualInput;
  END_VAR

  IF StrPh.run AND NOT StrPh.start THEN
  	StrPh.start := TRUE;
  	StrPh.top := FALSE;
  	StrPh.error := FALSE;
            StrPh.run:=FALSE;
  END_IF;

  IF StrPh.top THEN StrPh.error := FALSE; END_IF;

  reset_Trig(CLK := StrPh.reset);
  IF reset_Trig.Q THEN
  	StrPh.start := FALSE;
  	StrPh.error := FALSE;
  	StrPh.top := FALSE;
            StrPh.run:=FALSE;
            StrPh.reset:=FALSE;
  END_IF;

  StrPh.startStatus := SHL(BOOL_TO_DWORD(StrPh.start), PhaseNumber);
  StrPh.errorStatus := SHL(BOOL_TO_DWORD(StrPh.error), PhaseNumber);
  StrPh.topStatus := SHL(BOOL_TO_DWORD(StrPh.top), PhaseNumber);
END_FUNCTION_BLOCK

FUNCTION runPhase : BOOL
  VAR_IN_OUT
    ph : struct_PhaseAlgoritm;
  END_VAR

  IF NOT ph.start THEN
                      ph.run:=TRUE;
  END_IF;
END_FUNCTION

FUNCTION resetPhase : BOOL
  VAR_IN_OUT
    ph : struct_PhaseAlgoritm;
  END_VAR

  IF ph.start OR ph.top THEN
                      ph.reset:=TRUE;
  END_IF;
END_FUNCTION

FUNCTION askQuestion : BOOL
  VAR_IN_OUT
    StrQ : struct_Question;
  END_VAR

  IF NOT StrQ.ask THEN
                      StrQ.inOpcCommandsDisabled:=FALSE;
                      StrQ.ask:=TRUE;
  END_IF;
END_FUNCTION

FUNCTION resetQuestion : BOOL
  VAR_IN_OUT
    StrQ : struct_Question;
  END_VAR

  IF StrQ.ask THEN
                      StrQ.inOpcCommandsDisabled:=TRUE;
                      StrQ.reset:=TRUE;
  END_IF;
END_FUNCTION

FUNCTION_BLOCK fb_vibegPNSAlg
  VAR_IN_OUT
    StrAlg : struct_Alg;
  END_VAR
  VAR
    autoPnsOff : struct_PhaseAlgoritm;
    waitVibeg : struct_PhaseAlgoritm;
    pnsOff : struct_PhaseAlgoritm;
    vibegEnd : struct_PhaseAlgoritm;
  END_VAR
  VAR_IN_OUT
    algContinue : struct_Question;
  END_VAR
  VAR
    fb_autoPnsOff : fb_ph_algoritm;
    fb_waitVibeg : fb_ph_Timer;
    fb_algContinue : fb_Question;
    fb_pnsOff : fb_ph_Switch;
    fb_vibegEnd : fb_ph_CustomPhase;
    _sunpackerCommand : fb_sunpackerCommand;
    _statusAi : TYPE_StatusAi;
    _Answers : TYPE_Answers;
    _statusDualInput : TYPE_statusDualInput;
    _DualStateImAction : TYPE_DualStateImAction;
    _PhaseAlgoritmAction : TYPE_PhaseAlgoritmAction;
    source : BYTE;
    cmd : BYTE;
    lastCmd : BYTE;
    source_for_Status : BYTE;
    cmd_for_Status : BYTE;
    command_error_for_Status : BYTE;
    resetCmdTimer : TON;
    resetCmdTimerPriznak : BOOL;
    onInit : BOOL;
    waitReset : TON;
  END_VAR
  VAR_EXTERNAL
    IM : ImConfig;
    algoritms : AlgoritmsConfig;
    ai : AiConfig;
    protections : ProtectionsConfig;
    AlgTimers : struct_AlgTimers;
  END_VAR

  IF NOT onInit THEN
   fb_autoPnsOff(phaseNumber:=0, act:=_reset, waitCompletion:=FALSE);
    fb_waitVibeg(phaseNumber:=1, delay:=T#300S);
       algContinue.AnswerVariants:=_Answers.ANS_YES;
       fb_pnsOff(phaseNumber:=2, act:=_off);
     fb_vibegEnd(phaseNumber:=14);
  onInit:=TRUE;
  END_IF;

   fb_autoPnsOff(StrPh:=autoPnsOff, alg:=algoritms.autoPns);
    fb_waitVibeg(StrPh:=waitVibeg, timer:=AlgTimers.vibegPNS_Timer);
  fb_algContinue(StrQ:=algContinue);
       fb_pnsOff(StrPh:=pnsOff, Im:=IM.pns);
     fb_vibegEnd(StrPh:=vibegEnd);

  IF StrAlg.isRuning THEN

  StrAlg.hasError := autoPnsOff.error OR pnsOff.error;

      IF IM.pns.onStatus = _statusDualInput.STATUS_ON AND NOT vibegEnd.top THEN

  	runPhase(vibegEnd);
            runPhase(waitVibeg);
            askQuestion(algContinue);

      END_IF;

      IF waitVibeg.top OR (algContinue.answer = _Answers.ANS_YES) THEN
  	vibegEnd.top:=TRUE;
  	resetPhase(waitVibeg);
            resetQuestion(algContinue);

            resetAiProtection(protections.P_masla_smazki_nizkoe_LA);
            resetDiProtection(protections.DavlenieMaslaSmazkiDi);

  	IM.SingleSignals.P_oil_low.Disabled_Sig:=TRUE;
  	ai.P_masla_smazki_nizkoe.Disabled_LA:=TRUE;
            ai.P_masla_smazki_nizkoe.Disabled_LW:=TRUE;
            ai.P_masla_smazki_srednee_posle_nasosov.Disabled_LW:=TRUE;
  	runPhase(pnsOff);
      END_IF;

      StrAlg.isEnded:=pnsOff.top;

  END_IF;

  StrAlg.CanRun := StrAlg.inCanRun;
  StrAlg.OpcCommandsDisabled := StrAlg.inOpcCommandsDisabled;

  (* ---- Если управление с ВУ заблокировано, то  передаем команду из алгоритма ---- *)
  IF StrAlg.inOpcCommandsDisabled THEN
  	StrAlg.inCommand := StrAlg.inCommand_Alg;
  ELSE (* иначе передаем команду с АРМа*)
  	StrAlg.inCommand := StrAlg.inCommand_ARM;
  END_IF;

  _sunpackerCommand(command := StrAlg.inCommand);
  	source := _sunpackerCommand.source;
  	cmd := _sunpackerCommand.cmd;

  IF cmd <> 0 AND lastCmd <> cmd AND (((NOT StrAlg.opcCommandsDisabled) AND source > 0) OR source = 0) then
  	CASE BYTE_TO_INT(cmd) OF
  		(*cmdRun*) 1: 	IF (StrAlg.CanRun) THEN
  					StrAlg.isRuning := TRUE;
  					StrAlg.isEnded := FALSE;
  					StrAlg.hasError := FALSE;
  					(*****************       OnRun       *****************)
                                                    runPhase(autoPnsOff);

  					cmd_for_Status := cmd;
  					source_for_Status := source;
  					command_error_for_Status := 0;
  				ELSE
  					StrAlg.isRuning := FALSE;
  					StrAlg.isEnded := FALSE;
  					StrAlg.hasError 	:= FALSE;

  					cmd_for_Status := 0;
  					source_for_Status := source;
  					command_error_for_Status := cmd;
  				END_IF;
  		(*cmdReset*) 2: 	StrAlg.isRuning := FALSE;
  				StrAlg.isEnded := FALSE;
  				StrAlg.hasError 	:= FALSE;

                                           (*****************       OnReset       *****************)
                                         waitReset(IN:=FALSE);
                                         resetPhase(autoPnsOff);
                                         resetPhase(waitVibeg);
                                         resetPhase(vibegEnd);
                                         resetPhase(pnsOff);
                                         resetQuestion(algContinue);

  				cmd_for_Status := cmd;
  				source_for_Status := source;
  				command_error_for_Status := 0;
  	END_CASE;
  	resetCmdTimer(IN := false);
  	resetCmdTimerPriznak := TRUE;
  END_IF;
  lastCmd := cmd;

  resetCmdTimer(IN := resetCmdTimerPriznak, PT := T#5S);
  IF resetCmdTimer.Q THEN
  	resetCmdTimerPriznak := FALSE;
  	source_for_Status := 0;
  	cmd_for_Status := 0;
  	command_error_for_Status := 0;
  END_IF;

  StrAlg.Start:= autoPnsOff.startStatus
              OR waitVibeg.startStatus
              OR pnsOff.startStatus
              OR vibegEnd.startStatus;

  StrAlg.Error:= autoPnsOff.errorStatus
              OR waitVibeg.errorStatus
              OR pnsOff.errorStatus
              OR vibegEnd.errorStatus;

  StrAlg.Top:=   autoPnsOff.topStatus
              OR waitVibeg.topStatus
              OR pnsOff.topStatus
              OR vibegEnd.topStatus;

  (*TODO: TYPE PROGRAM CODE HERE*)
  StrAlg.status :=  SHL(BYTE_TO_DWORD(source_for_Status), 29)
  			OR SHL(BYTE_TO_DWORD(cmd_for_Status), 26)
  			OR SHL(BYTE_TO_DWORD(command_error_for_Status), 23)
  			OR SHL(BOOL_TO_DWORD(StrAlg.OpcCommandsDisabled ), 21)
  			OR SHL(BOOL_TO_DWORD(StrAlg.hasError),4)
  			OR SHL(BOOL_TO_DWORD(StrAlg.CanRun),2)
  			OR SHL(BOOL_TO_DWORD(StrAlg.isEnded),1)
  			OR BOOL_TO_DWORD(StrAlg.isRuning);
END_FUNCTION_BLOCK

FUNCTION setValue : BOOL
  VAR_IN_OUT
    StrDP : struct_DiscretParametr;
  END_VAR
  VAR_INPUT
    newValue : UINT;
  END_VAR
  VAR
    cmd_ChangeValue : WORD := 1;
  END_VAR

  StrDP.newValue:=newValue;
  StrDP.inOpcCommandsDisabled:=TRUE;
  StrDP.inCommand_Alg:=cmd_ChangeValue;
END_FUNCTION

FUNCTION_BLOCK fb_AutoNUAlg
  VAR_IN_OUT
    StrAlg : struct_Alg;
    nu1 : struct_OilPump;
    nu2 : struct_OilPump;
  END_VAR
  VAR_INPUT
    dPoil : struct_AI;
  END_VAR
  VAR_IN_OUT
    mainNU : struct_DiscretParametr;
    Lowdp_di : struct_singleSignal;
    Ust_Swap : struct_AnalogParametr;
  END_VAR
  VAR
    _prevMainNU : UINT;
    _sunpackerCommand : fb_sunpackerCommand;
    _statusAi : TYPE_StatusAi;
    _statusDualInput : TYPE_statusDualInput;
    _commandDualInput : TYPE_commandDualInput;
    source : BYTE;
    cmd : BYTE;
    lastCmd : BYTE;
    source_for_Status : BYTE;
    cmd_for_Status : BYTE;
    command_error_for_Status : BYTE;
    resetCmdTimer : TON;
    waitPressure : TON;
    waitPressureTrig : R_TRIG;
    resetCmdTimerPriznak : BOOL;
    onInit : BOOL;
    onStart : BOOL;
  END_VAR
  VAR_EXTERNAL
    NotHasRezervNU : BOOL;
    Reset_HasNU : BOOL;
  END_VAR

  IF NOT onInit THEN
  StrAlg.inCanRun:=TRUE;
  StrAlg.inOpcCommandsDisabled:=TRUE;
  (*nu1.Osnovnoy:=TRUE; nu2.Osnovnoy:=FALSE;*)
  onInit:=TRUE;
  END_IF;

  IF Reset_HasNU THEN
  nu1.inBlocked:=FALSE;
  nu2.inBlocked:=FALSE;
  END_IF;

  NotHasRezervNU:=(nu1.Blocked OR nu2.Blocked);

  IF StrAlg.isRuning THEN

  StrAlg.hasError := nu1.CommandFault OR nu2.CommandFault OR (dPoil.interval<_statusAi.normal);

   IF mainNU.value<>_prevMainNU OR NOT onStart THEN

          CASE mainNU.value OF
  	0: nu1.Osnovnoy:=TRUE; nu2.Osnovnoy:=FALSE;
  	1: nu1.Osnovnoy:=FALSE; nu2.Osnovnoy:=TRUE;

          END_CASE;

      IF  nu1.Osnovnoy AND NOT nu1.Blocked THEN
          nu1.inCommand_Alg:=BYTE_TO_WORD(_commandDualInput.CMD_ON);
      ELSIF NOT NotHasRezervNU THEN
          nu1.inCommand_Alg:=BYTE_TO_WORD(_commandDualInput.CMD_OFF);
      END_IF;

      IF  nu2.Osnovnoy AND NOT nu2.Blocked THEN
          nu2.inCommand_Alg:=BYTE_TO_WORD(_commandDualInput.CMD_ON);
       ELSIF NOT NotHasRezervNU THEN
          nu2.inCommand_Alg:=BYTE_TO_WORD(_commandDualInput.CMD_OFF);
      END_IF;
        onStart:=TRUE;
       _prevMainNU:=mainNU.value;
   END_IF;

    (*IF (nu1.onStatus = _statusDualInput.STATUS_On) OR (nu2.onStatus = _statusDualInput.STATUS_On) THEN*)
      (*Если через 5С насос не нагнал 100кПа масла - он сломался и надо переключить насос*)
      IF dPoil.interval>= _statusAi.NORMAL THEN
            waitPressure(IN:=(dPoil.value<Ust_Swap.Value OR LowdP_DI.q) AND NOT NotHasRezervNU, PT:= T#5S);
      ELSE
  	waitPressure(IN:=(FALSE));
      END_IF;

      waitPressureTrig(CLK:=waitPressure.Q);
      IF waitPressureTrig.Q THEN
  	(*IF nu1.onStatus = _statusDualInput.STATUS_ON THEN*)
             IF mainNU.value = 0 THEN
  		nu1.inBlocked:=TRUE;
                      nu1.inCommand_Alg:=BYTE_TO_WORD(_commandDualInput.CMD_OFF);
  			(*IF 	mainNU.value = 0 THEN*)
                                          setValue(mainNU, 1);
  			(*END_IF;*)
  	END_IF;

  	(*IF nu2.onStatus = _statusDualInput.STATUS_ON THEN*)
            IF mainNU.value = 1 THEN
  		nu2.inBlocked:=TRUE;
                      nu2.inCommand_Alg:=BYTE_TO_WORD(_commandDualInput.CMD_OFF);
  			(*IF 	mainNU.value = 1 THEN*)
  				setValue(mainNU, 0);
  			(*END_IF;*)
  	END_IF;
      END_IF;
   (* END_IF;*)

  END_IF;

  StrAlg.CanRun := StrAlg.inCanRun;

  StrAlg.OpcCommandsDisabled := StrAlg.inOpcCommandsDisabled;

  (* ---- Если управление с ВУ заблокировано, то  передаем команду из алгоритма ---- *)
  IF StrAlg.inOpcCommandsDisabled THEN
  	StrAlg.inCommand := StrAlg.inCommand_Alg;
  ELSE (* иначе передаем команду с АРМа*)
  	StrAlg.inCommand := StrAlg.inCommand_ARM;
  END_IF;

  _sunpackerCommand(command := StrAlg.inCommand);
  	source := _sunpackerCommand.source;
  	cmd := _sunpackerCommand.cmd;

  IF cmd <> 0 AND lastCmd <> cmd AND (((NOT StrAlg.opcCommandsDisabled) AND source > 0) OR source = 0) then
  	CASE BYTE_TO_INT(cmd) OF
  		(*cmdRun*) 1: 	IF (StrAlg.CanRun) THEN
  					StrAlg.isRuning := TRUE;
  					StrAlg.isEnded := FALSE;
  					StrAlg.hasError := FALSE;

                                                    (*****************       OnRun       *****************)
  					nu1.inOpcCommandsDisabled:=TRUE;
                                                    nu2.inOpcCommandsDisabled:=TRUE;

  					cmd_for_Status := cmd;
  					source_for_Status := source;
  					command_error_for_Status := 0;
  				ELSE
  					StrAlg.isRuning := FALSE;
  					StrAlg.isEnded := FALSE;
  					StrAlg.hasError 	:= FALSE;

  					cmd_for_Status := 0;
  					source_for_Status := source;
  					command_error_for_Status := cmd;
  				END_IF;
  		(*cmdReset*) 2: 	StrAlg.isRuning := FALSE;
  				StrAlg.isEnded := FALSE;
  				StrAlg.hasError 	:= FALSE;

                                          (*****************       OnReset       *****************)
                                          waitPressure(IN:=(FALSE));
                                          onStart:=FALSE;

  				cmd_for_Status := cmd;
  				source_for_Status := source;
  				command_error_for_Status := 0;
  	END_CASE;
  	resetCmdTimer(IN := false);
  	resetCmdTimerPriznak := TRUE;
  END_IF;
  lastCmd := cmd;

  resetCmdTimer(IN := resetCmdTimerPriznak, PT := T#5S);
  IF resetCmdTimer.Q THEN
  	resetCmdTimerPriznak := FALSE;
  	source_for_Status := 0;
  	cmd_for_Status := 0;
  	command_error_for_Status := 0;
  END_IF;

  (*TODO: TYPE PROGRAM CODE HERE*)
  StrAlg.status :=  SHL(BYTE_TO_DWORD(source_for_Status), 29)
  			OR SHL(BYTE_TO_DWORD(cmd_for_Status), 26)
  			OR SHL(BYTE_TO_DWORD(command_error_for_Status), 23)
  			OR SHL(BOOL_TO_DWORD(StrAlg.OpcCommandsDisabled ), 21)
                                OR SHL(BOOL_TO_DWORD(NotHasRezervNU), 15)
  			OR SHL(BOOL_TO_DWORD(StrAlg.hasError),4)
  			OR SHL(BOOL_TO_DWORD(StrAlg.CanRun),2)
  			OR SHL(BOOL_TO_DWORD(StrAlg.isEnded),1)
  			OR BOOL_TO_DWORD(StrAlg.isRuning);
END_FUNCTION_BLOCK

FUNCTION_BLOCK fb_ph_WaitAnalogValue
  VAR_IN_OUT
    ai : struct_AI;
  END_VAR
  VAR_INPUT
    more : LREAL;
    less : LREAL;
    PhaseNumber : UINT;
  END_VAR
  VAR_IN_OUT
    StrPh : struct_PhaseAlgoritm;
  END_VAR
  VAR
    CommandFault_Trig : R_TRIG;
    reset_Trig : R_TRIG;
    _statusAi : TYPE_StatusAi;
    _statusDualInput : TYPE_statusDualInput;
  END_VAR

  IF StrPh.run AND NOT StrPh.start THEN
  	StrPh.start := TRUE;
  	StrPh.top := FALSE;
  	StrPh.error := FALSE;
            StrPh.run:=FALSE;
  END_IF;

  IF StrPh.start AND NOT StrPh.top THEN
                      IF ai.interval < _statusAi.normal THEN
  	              StrPh.error := TRUE;
                          StrPh.top:=FALSE;
                      ELSE
                              IF (more<>0.0) OR (less<>0.0) THEN
                              StrPh.top:=TRUE;
  	                    IF more<>0.0 THEN StrPh.top:=StrPh.top AND (ai.value > more); END_IF;
  	                    IF less<>0.0 THEN StrPh.top:=StrPh.top AND (ai.value < less); END_IF;
                              ELSE
  	                  StrPh.top:=TRUE;
                              END_IF;
                     END_IF;
  END_IF;

  IF StrPh.top THEN
  StrPh.error := FALSE;
  END_IF;

  reset_Trig(CLK := StrPh.reset);
  IF reset_Trig.Q THEN
  	StrPh.start := FALSE;
  	StrPh.error := FALSE;
  	StrPh.top := FALSE;
            StrPh.run:=FALSE;
            StrPh.reset:=FALSE;
  END_IF;

  StrPh.startStatus := SHL(BOOL_TO_DWORD(StrPh.start), PhaseNumber);
  StrPh.errorStatus := SHL(BOOL_TO_DWORD(StrPh.error), PhaseNumber);
  StrPh.topStatus := SHL(BOOL_TO_DWORD(StrPh.top), PhaseNumber);
END_FUNCTION_BLOCK

FUNCTION_BLOCK fb_ph_OilPump
  VAR_IN_OUT
    im : struct_OilPump;
  END_VAR
  VAR_INPUT
    act : TYPE_DualStateImAction;
    PhaseNumber : UINT;
  END_VAR
  VAR_IN_OUT
    StrPh : struct_PhaseAlgoritm;
  END_VAR
  VAR
    CommandFault_Trig : R_TRIG;
    reset_Trig : R_TRIG;
    _statusDualInput : TYPE_statusDualInput;
  END_VAR

  IF StrPh.run AND NOT StrPh.start THEN
  	StrPh.start := TRUE;
  	StrPh.top := FALSE;
  	StrPh.error := FALSE;

  	CASE act OF
  		(*DualStateImAction.on*)   _on :im.inOpcCommandsDisabled:=TRUE;
                                                      im.inCommand_Alg := 1; (*cmd_open*)
  		(*DualStateImAction.off*) _off :im.inOpcCommandsDisabled:=TRUE;
                                                      im.inCommand_Alg := 2; (*cmd_close*)
  	END_CASE;
  END_IF;

  IF StrPh.start OR StrPh.reset THEN
      StrPh.run:=FALSE;
  END_IF;

  IF StrPh.start AND NOT StrPh.top THEN
                      CommandFault_Trig(CLK := im.CommandFault);
                      IF CommandFault_Trig.Q THEN
  	          StrPh.error := TRUE;
                      END_IF;

  		CASE act OF
  		(*_DualStateImAction.on*)    _on: StrPh.top := im.onStatus = _statusDualInput.STATUS_ON;
  		(*_DualStateImAction.off*)  _off: StrPh.top := im.onStatus = _statusDualInput.STATUS_OFF;
  		END_CASE;

  END_IF;

  reset_Trig(CLK := StrPh.reset);
  IF reset_Trig.Q THEN
  	StrPh.start := FALSE;
  	StrPh.error := FALSE;
  	StrPh.top := FALSE;
            StrPh.reset:=FALSE;
  END_IF;

  StrPh.startStatus := SHL(BOOL_TO_DWORD(StrPh.start), PhaseNumber);
  StrPh.errorStatus := SHL(BOOL_TO_DWORD(StrPh.error), PhaseNumber);
  StrPh.topStatus := SHL(BOOL_TO_DWORD(StrPh.top), PhaseNumber);
END_FUNCTION_BLOCK

FUNCTION resetAndDisable : BOOL
  VAR_IN_OUT
    alg : struct_Alg;
  END_VAR
  VAR CONSTANT
    cmdReset : WORD := 2;
  END_VAR

  IF alg.isRuning THEN
                      alg.inOpcCommandsDisabled:=TRUE;
  		alg.inCommand_Alg:=cmdReset;
  END_IF;

   alg.inCanRun:=FALSE;
END_FUNCTION

FUNCTION runDiProtection : BOOL
  VAR_IN_OUT
    protection : struct_DiProtection;
  END_VAR
  VAR CONSTANT
    cmdRun : WORD := 1;
  END_VAR

  IF NOT protection.isRunning THEN
                      protection.inOpcCommandsDisabled:=TRUE;
  		protection.inCommand_Alg:=cmdRun;
  END_IF;
END_FUNCTION

FUNCTION runAiProtection : BOOL
  VAR_IN_OUT
    protection : struct_AiProtection;
  END_VAR
  VAR CONSTANT
    cmdRun : WORD := 1;
  END_VAR

  IF NOT protection.isRunning THEN
                      protection.inOpcCommandsDisabled:=TRUE;
  		protection.inCommand_Alg:=cmdRun;
  END_IF;
END_FUNCTION

FUNCTION_BLOCK fb_puskOilSystemAlg
  VAR_IN_OUT
    StrAlg : struct_Alg;
  END_VAR
  VAR
    pnsOn : struct_PhaseAlgoritm;
    LowOil : struct_PhaseAlgoritm;
    BreakPuskTimer_Poil : struct_PhaseAlgoritm;
    Poil_DefenseActive : struct_PhaseAlgoritm;
    autoNuOn : struct_PhaseAlgoritm;
    nuOn : struct_PhaseAlgoritm;
    nu1On : struct_PhaseAlgoritm;
    nu2On : struct_PhaseAlgoritm;
    di_dPmg : struct_PhaseAlgoritm;
    dP_oilGas100 : struct_PhaseAlgoritm;
    runProtect_dP : struct_PhaseAlgoritm;
    testUnsuccessful : struct_PhaseAlgoritm;
    fb_pnsOn : fb_ph_Switch;
    fb_LowOil : fb_ph_WaitAnalogValue;
    fb_BreakPuskTimer_Poil : fb_ph_Timer;
    fb_Poil_DefenseActive : fb_ph_CustomPhase;
    fb_nuOn : fb_ph_CustomPhase;
    fb_nu1On : fb_ph_OilPump;
    fb_nu2On : fb_ph_OilPump;
    fb_autoNuOn : fb_ph_algoritm;
    fb_di_dPmg : fb_ph_CustomPhase;
    fb_dP_oilGas100 : fb_ph_WaitAnalogValue;
    fb_runProtect_dP : fb_ph_CustomPhase;
    fb_testUnsuccessful : fb_ph_CustomPhase;
    _sunpackerCommand : fb_sunpackerCommand;
    _statusAi : TYPE_StatusAi;
    _Answers : TYPE_Answers;
    _statusDualInput : TYPE_statusDualInput;
    _DualStateImAction : TYPE_DualStateImAction;
    _PhaseAlgoritmAction : TYPE_PhaseAlgoritmAction;
    source : BYTE;
    cmd : BYTE;
    lastCmd : BYTE;
    source_for_Status : BYTE;
    cmd_for_Status : BYTE;
    command_error_for_Status : BYTE;
    resetCmdTimer : TON;
    resetCmdTimerPriznak : BOOL;
    onInit : BOOL;
    waitReset : TON;
  END_VAR
  VAR_EXTERNAL
    IM : ImConfig;
    algoritms : AlgoritmsConfig;
    ai : AiConfig;
    protections : ProtectionsConfig;
    AlgTimers : struct_AlgTimers;
  END_VAR

  IF NOT onInit THEN
                 fb_pnsOn(phaseNumber:=0, act:=_on);
                fb_LowOil(phaseNumber:=1);
   fb_BreakPuskTimer_Poil(phaseNumber:=3, delay:=T#240S);
    fb_Poil_DefenseActive(phaseNumber:=5);
                  fb_nuOn(phaseNumber:=6);
                 fb_nu1On(phaseNumber:=11, act:=_on);
                 fb_nu2On(phaseNumber:=12, act:=_on);
              fb_autoNuOn(phaseNumber:=7, act:=_run, waitCompletion:=FALSE);
               fb_di_dPmg(phaseNumber:=8);
          fb_dP_oilGas100(phaseNumber:=9);
         fb_runProtect_dP(phaseNumber:=10);
      fb_testUnsuccessful(phaseNumber:=17);

  onInit:=TRUE;
  END_IF;

                fb_pnsOn(StrPh:=pnsOn, Im:=IM.pns);
               fb_LowOil(StrPh:=LowOil, ai:=ai.P_masla_smazki_nizkoe, more:=im.AutoPns_UstRun.Value);
  fb_BreakPuskTimer_Poil(StrPh:=BreakPuskTimer_Poil, timer:=AlgTimers.puskOilSystem_BreakPuskTimer_Poil);
   fb_Poil_DefenseActive(StrPh:=Poil_DefenseActive);
                 fb_nuOn(StrPh:=nuOn);
                fb_nu1On(StrPh:=nu1On, Im:=Im.nu1);
                fb_nu2On(StrPh:=nu2On, Im:=Im.nu2);
             fb_autoNuOn(StrPh:=autoNuOn, alg:=algoritms.autoNu);
              fb_di_dPmg(StrPh:=di_dPmg);
         fb_dP_oilGas100(StrPh:=dP_oilGas100, ai:=ai.dPmaslo_gaz, more:=im.PuskOilSystem_UstdPmg.Value);
        fb_runProtect_dP(StrPh:=runProtect_dP);
     fb_testUnsuccessful(StrPh:=testUnsuccessful);

  IF StrAlg.isRuning THEN

      StrAlg.hasError := LowOil.error OR dP_oilGas100.error OR pnsOn.error OR testUnsuccessful.error;

      IF pnsOn.top THEN
          runPhase(LowOil);
      END_IF;

      IF LowOil.top THEN
          runAiProtection(protections.P_masla_smazki_nizkoe_LA);
          runDiProtection(protections.DavlenieMaslaSmazkiDi);
          runPhase(Poil_DefenseActive);
          IM.SingleSignals.P_oil_low.Disabled_Sig:=FALSE;
          ai.P_masla_smazki_nizkoe.Disabled_LA:=FALSE;
          ai.P_masla_smazki_nizkoe.Disabled_LW:=FALSE;
          ai.P_masla_smazki_srednee_posle_nasosov.Disabled_LW:=FALSE;
      END_IF;

      IF Poil_DefenseActive.start AND NOT Poil_DefenseActive.top THEN
         Poil_DefenseActive.top:=protections.P_masla_smazki_nizkoe_LA.isRunning AND protections.DavlenieMaslaSmazkiDi.isRunning;
      END_IF;

      IF Poil_DefenseActive.top THEN
         (* runPhase(autoNuOn);*)
  	runPhase(nuOn);
      END_IF;

      IF nuOn.start AND NOT nuOn.top THEN
          IF IM.AutoNU_mainNU.Value = 0 THEN
              runPhase(nu1On);
          END_IF;

          IF IM.AutoNU_mainNU.Value = 1 THEN
              runPhase(nu2On);
          END_IF;
         nuOn.top:= Im.nu1.onStatus = _statusDualInput.STATUS_ON OR Im.nu2.onStatus = _statusDualInput.STATUS_ON;
      END_IF;

      IF nuOn.top THEN
  	runPhase(di_dPmg);
            runPhase(dP_oilGas100);
      END_IF;

      IF di_dPmg.start AND NOT di_dPmg.top THEN
         di_dPmg.top:= NOT IM.SingleSignals.dP_oilgaz_low.Q;
      END_IF;

      IF dP_oilGas100.top AND di_dPmg.top THEN
            runPhase(autoNuOn);
  	runPhase(runProtect_dP);
  	runAiProtection(protections.dP_maslogaz_LA);
            runDiProtection(protections.dP_masloGaz_LowDI);
            IM.SingleSignals.dP_oilgaz_low.Disabled_Sig:=FALSE;
            ai.dPmaslo_gaz.Disabled_LA:=FALSE;
            ai.dPmaslo_gaz.Disabled_LW:=FALSE;
      END_IF;

      IF runProtect_dP.start AND NOT runProtect_dP.top THEN
         runProtect_dP.top:= protections.dP_maslogaz_LA.isRunning AND protections.dP_masloGaz_LowDI.isRunning;
      END_IF;

      IF BreakPuskTimer_Poil.top AND (NOT runProtect_dP.top) THEN
  	testUnsuccessful.error:=TRUE;
      END_IF;

      IF runProtect_dP.top THEN
            resetPhase(BreakPuskTimer_Poil);
  	waitReset(IN:=TRUE);
      END_IF;

      IF waitReset.Q AND NOT (algoritms.Apusk.isRuning OR algoritms.SemiAutoPusk.isRuning) THEN
      resetAndDisable(StrAlg);
      END_IF;

      StrAlg.isEnded:=runProtect_dP.top;
  END_IF;

  StrAlg.CanRun := StrAlg.inCanRun;
  StrAlg.OpcCommandsDisabled := StrAlg.inOpcCommandsDisabled;

  (* ---- Если управление с ВУ заблокировано, то  передаем команду из алгоритма ---- *)
  IF StrAlg.inOpcCommandsDisabled THEN
  	StrAlg.inCommand := StrAlg.inCommand_Alg;
  ELSE (* иначе передаем команду с АРМа*)
  	StrAlg.inCommand := StrAlg.inCommand_ARM;
  END_IF;

  _sunpackerCommand(command := StrAlg.inCommand);
  	source := _sunpackerCommand.source;
  	cmd := _sunpackerCommand.cmd;

  IF cmd <> 0 AND lastCmd <> cmd AND (((NOT StrAlg.opcCommandsDisabled) AND source > 0) OR source = 0) then
  	CASE BYTE_TO_INT(cmd) OF
  		(*cmdRun*) 1: 	IF (StrAlg.CanRun) THEN
  					StrAlg.isRuning := TRUE;
  					StrAlg.isEnded := FALSE;
  					StrAlg.hasError := FALSE;
  					(*****************       OnRun       *****************)
                                                    runPhase(pnsOn);
                                                    runPhase(BreakPuskTimer_Poil);
                                                    runPhase(testUnsuccessful);
  					cmd_for_Status := cmd;
  					source_for_Status := source;
  					command_error_for_Status := 0;
  				ELSE
  					StrAlg.isRuning := FALSE;
  					StrAlg.isEnded := FALSE;
  					StrAlg.hasError 	:= FALSE;

  					cmd_for_Status := 0;
  					source_for_Status := source;
  					command_error_for_Status := cmd;
  				END_IF;
  		(*cmdReset*) 2: 	StrAlg.isRuning := FALSE;
  				StrAlg.isEnded := FALSE;
  				StrAlg.hasError 	:= FALSE;

                                           (*****************       OnReset       *****************)
                                          waitReset(IN:=FALSE);
                                          resetPhase(pnsOn);
                                          resetPhase(LowOil);
                                          resetPhase(BreakPuskTimer_Poil);
                                          resetPhase(Poil_DefenseActive);
                                          resetPhase(autoNuOn);
                                          resetPhase(nu1On);
                                          resetPhase(nu2On);
                                          resetPhase(nuOn);
                                          resetPhase(di_dPmg);
                                          resetPhase(dP_oilGas100);
                                          resetPhase(runProtect_dP);
                                          resetPhase(testUnsuccessful);
  	                              (*protections.P_masla_smazki_nizkoe_LA.inOpcCommandsDisabled:=FALSE;
                                          protections.DavlenieMaslaSmazkiDi.inOpcCommandsDisabled:=FALSE;
                                          protections.dP_maslogaz_LA.inOpcCommandsDisabled:=FALSE;
                                          protections.dP_masloGaz_LowDI.inOpcCommandsDisabled:=FALSE;*)

  				cmd_for_Status := cmd;
  				source_for_Status := source;
  				command_error_for_Status := 0;
  	END_CASE;
  	resetCmdTimer(IN := false);
  	resetCmdTimerPriznak := TRUE;
  END_IF;
  lastCmd := cmd;

  resetCmdTimer(IN := resetCmdTimerPriznak, PT := T#5S);
  IF resetCmdTimer.Q THEN
  	resetCmdTimerPriznak := FALSE;
  	source_for_Status := 0;
  	cmd_for_Status := 0;
  	command_error_for_Status := 0;
  END_IF;

  StrAlg.Start:= pnsOn.startStatus
              OR LowOil.startStatus
              OR BreakPuskTimer_Poil.startStatus
              OR Poil_DefenseActive.startStatus
              OR nuOn.startStatus
              OR di_dPmg.startStatus
              OR dP_oilGas100.startStatus
              OR runProtect_dP.startStatus
              OR testUnsuccessful.startStatus;

  StrAlg.Error:= pnsOn.errorStatus
              OR LowOil.errorStatus
              OR BreakPuskTimer_Poil.errorStatus
              OR Poil_DefenseActive.errorStatus
              OR nuOn.errorStatus
              OR di_dPmg.errorStatus
              OR dP_oilGas100.errorStatus
              OR runProtect_dP.errorStatus
              OR testUnsuccessful.errorStatus;

  StrAlg.Top:=   pnsOn.topStatus
              OR LowOil.topStatus
              OR BreakPuskTimer_Poil.topStatus
              OR Poil_DefenseActive.topStatus
              OR nuOn.topStatus
              OR di_dPmg.topStatus
              OR dP_oilGas100.topStatus
              OR runProtect_dP.topStatus
              OR testUnsuccessful.topStatus;

  (*TODO: TYPE PROGRAM CODE HERE*)
  StrAlg.status :=  SHL(BYTE_TO_DWORD(source_for_Status), 29)
  			OR SHL(BYTE_TO_DWORD(cmd_for_Status), 26)
  			OR SHL(BYTE_TO_DWORD(command_error_for_Status), 23)
  			OR SHL(BOOL_TO_DWORD(StrAlg.OpcCommandsDisabled ), 21)
  			OR SHL(BOOL_TO_DWORD(StrAlg.hasError),4)
  			OR SHL(BOOL_TO_DWORD(StrAlg.CanRun),2)
  			OR SHL(BOOL_TO_DWORD(StrAlg.isEnded),1)
  			OR BOOL_TO_DWORD(StrAlg.isRuning);
END_FUNCTION_BLOCK

FUNCTION_BLOCK fb_TableValue_Min
  VAR_INPUT
    parametr : REAL;
  END_VAR
  VAR
    _table : ARRAY [0..8] OF TYPE_TableRec;
  END_VAR
  VAR_INPUT
    inverse : BOOL := FALSE;
  END_VAR
  VAR_IN_OUT
    actualValue : REAL;
  END_VAR
  VAR
    indexLess : INT := -1;
    indexMore : INT := -1;
  END_VAR
  VAR CONSTANT
    maxTableLength : INT := 9;
  END_VAR
  VAR
    Vali : REAL;
    i : INT;
    moreDistance : REAL;
    lessDistance : REAL;
    onInit : BOOL;
    _prevParam : REAL := 50.0;
  END_VAR

  IF NOT onInit THEN
  _table[0].x:=-35.0;  _table[0].y:=130.0;
  _table[1].x:=-25.0;  _table[1].y:=124.0;
  _table[2].x:=-15.0;  _table[2].y:=118.0;
  _table[3].x:= -5.0;  _table[3].y:=112.0;
  _table[4].x:=  0.0;  _table[4].y:=108.0;
  _table[5].x:=  5.0;  _table[5].y:=106.0;
  _table[6].x:= 15.0;  _table[6].y:=104.0;
  _table[7].x:= 25.0;  _table[7].y:=102.0;
  _table[8].x:= 35.0;  _table[8].y:= 97.0;

  onInit:=TRUE;
  END_IF;

  IF parametr <> _prevParam THEN
  indexLess:=-1;
  indexMore:=-1;
  lessDistance:=0.0;
  moreDistance:=0.0;
  FOR i:=0 TO maxTableLength-1 DO
  	IF NOT inverse THEN
  		Vali:=_table[i].x;
  	ELSE
  		Vali:=_table[i].y;
  	END_IF;

  	IF (Vali=parametr) THEN
  		indexLess:=i;
  		indexMore:=i;
  	ELSIF ((Vali<parametr) AND ((lessDistance>parametr-Vali) OR (indexLess<0))) THEN
  		indexLess:=i;
  		lessDistance:=parametr-Vali;
  	ELSIF ((Vali>parametr) AND ((moreDistance>Vali-parametr) OR (indexMore<0))) THEN
  		indexMore:=i;
  		moreDistance:=parametr-Vali;
  	END_IF;
  END_FOR;
  (*
  IF indexLess<0 THEN
  	indexLess:=indexMore;
  END_IF;

  IF indexMore<0 THEN
  	indexMore:=indexLess;
  END_IF;
  *)
    IF (_table[indexMore].x<>_table[indexLess].x) THEN
    actualValue:=_table[indexLess].y+((_table[indexMore].y-_table[indexLess].y)/(_table[indexMore].x-_table[indexLess].x))*(parametr-_table[indexLess].x);
    ELSE
    actualValue:=_table[indexLess].y;
    END_IF;
     _prevParam:= parametr;
  END_IF;
END_FUNCTION_BLOCK

FUNCTION_BLOCK fb_TableValue_Max
  VAR_INPUT
    parametr : REAL;
  END_VAR
  VAR
    _table : ARRAY [0..8] OF TYPE_TableRec;
  END_VAR
  VAR_INPUT
    inverse : BOOL := FALSE;
  END_VAR
  VAR_IN_OUT
    actualValue : REAL;
  END_VAR
  VAR
    indexLess : INT := -1;
    indexMore : INT := -1;
  END_VAR
  VAR CONSTANT
    maxTableLength : INT := 9;
  END_VAR
  VAR
    Vali : REAL;
    i : INT;
    moreDistance : REAL;
    lessDistance : REAL;
    onInit : BOOL;
    _prevParam : REAL := 50.0;
  END_VAR

  IF NOT onInit THEN
  _table[0].x:=-35.0;  _table[0].y:=320.0;
  _table[1].x:=-25.0;  _table[1].y:=315.0;
  _table[2].x:=-15.0;  _table[2].y:=310.0;
  _table[3].x:= -5.0;  _table[3].y:=305.0;
  _table[4].x:=  0.0;  _table[4].y:=300.0;
  _table[5].x:=  5.0;  _table[5].y:=295.0;
  _table[6].x:= 15.0;  _table[6].y:=290.0;
  _table[7].x:= 25.0;  _table[7].y:=285.0;
  _table[8].x:= 35.0;  _table[8].y:=280.0;

  onInit:=TRUE;
  END_IF;

  IF parametr <> _prevParam THEN
  indexLess:=-1;
  indexMore:=-1;
  lessDistance:=0.0;
  moreDistance:=0.0;
  FOR i:=0 TO maxTableLength-1 DO
  	IF NOT inverse THEN
  		Vali:=_table[i].x;
  	ELSE
  		Vali:=_table[i].y;
  	END_IF;

  	IF (Vali=parametr) THEN
  		indexLess:=i;
  		indexMore:=i;
  	ELSIF ((Vali<parametr) AND ((lessDistance>parametr-Vali) OR (indexLess<0))) THEN
  		indexLess:=i;
  		lessDistance:=parametr-Vali;
  	ELSIF ((Vali>parametr) AND ((moreDistance>Vali-parametr) OR (indexMore<0))) THEN
  		indexMore:=i;
  		moreDistance:=parametr-Vali;
  	END_IF;
  END_FOR;
  (*
  IF indexLess<0 THEN
  	indexLess:=indexMore;
  END_IF;

  IF indexMore<0 THEN
  	indexMore:=indexLess;
  END_IF;
  *)
    IF (_table[indexMore].x<>_table[indexLess].x) THEN
    actualValue:=_table[indexLess].y+((_table[indexMore].y-_table[indexLess].y)/(_table[indexMore].x-_table[indexLess].x))*(parametr-_table[indexLess].x);
    ELSE
    actualValue:=_table[indexLess].y;
    END_IF;
     _prevParam:= parametr;
  END_IF;
END_FUNCTION_BLOCK

FUNCTION_BLOCK fb_RashodAlg
  VAR_INPUT
    P_gasIn : struct_AI;
  END_VAR
  VAR_IN_OUT
    StrAi : struct_AI;
  END_VAR
  VAR_INPUT
    T_gasIn : struct_AI;
    dP_konf : struct_AI;
    K : struct_AnalogParametr;
    A : struct_AnalogParametr;
    y0 : struct_AnalogParametr;
  END_VAR
  VAR CONSTANT
    P0 : LREAL := 0.1033;
    T0 : LREAL := 293.0;
  END_VAR
  VAR
    num : LREAL;
    den : LREAL;
    _statusAi : TYPE_StatusAi;
  END_VAR

  strAI.opcCommandsDisabled := strAI.inopcCommandsDisabled ;

  IF (P_gasIn.interval < _statusAi.normal) OR
     (T_gasIn.interval < _statusAi.normal) OR
     (dP_konf.interval < _statusAi.normal) THEN
  	StrAi.interval := _statusAi.NOTRELIABLE;
            strAI.status := 	SHL(BOOL_TO_DWORD(strAI.OpcCommandsDisabled ), 21)
  	OR BYTE_TO_DWORD(strAI.interval);
  	RETURN;
  END_IF;

  IF (P_gasIn.value <0.3) THEN
  	StrAi.interval := _statusAi.normal;
  	StrAi.value:= 0.0;
            strAI.status := 	SHL(BOOL_TO_DWORD(strAI.OpcCommandsDisabled ), 21)
  	OR BYTE_TO_DWORD(strAI.interval);
  	RETURN;
  END_IF;

  StrAi.interval:= _statusAi.normal;

  num:= (dP_konf.Value/1000.0)*(T_gasIn.value+273.0)*P0*735.56*K.Value;
  den:= y0.Value*P_gasIn.value*T0 ;

  StrAi.value:= A.Value*SQRT(num/den);

  strAI.status := 	SHL(BOOL_TO_DWORD(strAI.OpcCommandsDisabled ), 21) (* Управление в ВУ заблокировано *)
  		OR BYTE_TO_DWORD(strAI.interval);	              (* интервал *)
END_FUNCTION_BLOCK

FUNCTION_BLOCK fb_ZapasAlg
  VAR_INPUT
    Q_actual : struct_AI;
  END_VAR
  VAR_IN_OUT
    StrAi : struct_AI;
  END_VAR
  VAR_INPUT
    Q_min : LREAL;
    Q_max : LREAL;
  END_VAR
  VAR
    _statusAi : TYPE_StatusAi;
  END_VAR

  IF (Q_actual.interval < _statusAi.normal) THEN
  	StrAi.interval := _statusAi.NOTRELIABLE;
            strAI.status := 	SHL(BOOL_TO_DWORD(strAI.OpcCommandsDisabled ), 21)
  		OR BYTE_TO_DWORD(strAI.interval);
  	RETURN;
  END_IF;

  IF (Q_actual.value <10.0) THEN
  	StrAi.interval := _statusAi.normal;
  	StrAi.value:= 100.0;
            strAI.status := 	SHL(BOOL_TO_DWORD(strAI.OpcCommandsDisabled ), 21)
  		OR BYTE_TO_DWORD(strAI.interval);
  	RETURN;
  END_IF;

  strAI.opcCommandsDisabled := strAI.inopcCommandsDisabled ;
  StrAi.interval:= _statusAi.normal;

  StrAi.value:= ((Q_actual.value - Q_min)/(Q_max-Q_min))*100.0;

  strAI.status := 	SHL(BOOL_TO_DWORD(strAI.OpcCommandsDisabled ), 21) (* Управление в ВУ заблокировано *)
  		OR BYTE_TO_DWORD(strAI.interval);	              (* интервал *)
END_FUNCTION_BLOCK

FUNCTION_BLOCK fb_AntiPompagAlg
  VAR
    tableQ_min : fb_TableValue_Min;
    tableQ_max : fb_TableValue_Max;
    fb_Rashod : fb_RashodAlg;
    fb_Zapas : fb_ZapasAlg;
  END_VAR
  VAR_IN_OUT
    Kran6 : struct_Kran;
    StrAlg : struct_Alg;
    Rashod : struct_AI;
    Zapas : struct_AI;
  END_VAR
  VAR_INPUT
    P_gasIn : struct_AI;
    T_gasIn : struct_AI;
    dP_konf : struct_AI;
    UgolVNA : struct_AnalogParametr;
    K : struct_AnalogParametr;
    A : struct_AnalogParametr;
    y0 : struct_AnalogParametr;
  END_VAR
  VAR
    Q_max : LREAL;
    Q_min : LREAL;
    pompaj : BOOL;
    _statusAi : TYPE_StatusAi;
    _statusDualInput : TYPE_statusDualInput;
    _sunpackerCommand : fb_sunpackerCommand;
    source : BYTE;
    cmd : BYTE;
    lastCmd : BYTE;
    source_for_Status : BYTE;
    cmd_for_Status : BYTE;
    command_error_for_Status : BYTE;
    resetCmdTimer : TON;
    resetCmdTimerPriznak : BOOL;
  END_VAR

  tableQ_min(parametr:=LREAL_TO_REAL(UgolVNA.Value));

  tableQ_max(parametr:=LREAL_TO_REAL(UgolVNA.Value));

  Q_min:=REAL_TO_LREAL(tableQ_min.actualValue);

  Q_max:=REAL_TO_LREAL(tableQ_max.actualValue);

  fb_Rashod(StrAi:=Rashod, P_gasIn:=P_gasIn, T_gasIn:=T_gasIn, dP_konf:=dP_konf, K:=K, A:=A, y0:=y0);

  fb_Zapas(StrAi:=Zapas, Q_actual:=Rashod, Q_min:=Q_min, Q_max:=Q_max);

  StrAlg.CanRun := StrAlg.inCanRun;

  StrAlg.OpcCommandsDisabled := StrAlg.inOpcCommandsDisabled;

  IF StrAlg.isRuning THEN

  StrAlg.hasError := (Rashod.interval < _statusAi.normal);

  pompaj:= (Rashod.interval>=_statusAi.normal) AND (Rashod.value <= Q_min);

  IF pompaj THEN
            Kran6.inOpcCommandsDisabled:=TRUE;
  	Kran6.inCommand_Alg := 1;  (*cmd_open*)
  END_IF;

  StrAlg.isEnded := Kran6.onStatus = _statusDualInput.STATUS_ON ;

  END_IF;

  (* ---- Если управление с ВУ заблокировано, то передаем команду из алгоритма ---- *)
  IF StrAlg.inOpcCommandsDisabled THEN
  	StrAlg.inCommand := StrAlg.inCommand_Alg;
  ELSE (* иначе передаем команду с АРМа*)
  	StrAlg.inCommand := StrAlg.inCommand_ARM;
  END_IF;

  _sunpackerCommand(command := StrAlg.inCommand);
  	source := _sunpackerCommand.source;
  	cmd := _sunpackerCommand.cmd;

  IF cmd <> 0 AND lastCmd <> cmd AND (((NOT StrAlg.opcCommandsDisabled) AND source > 0) OR source = 0) then
  	CASE BYTE_TO_INT(cmd) OF
  		(*cmdRun*) 1: 	IF (StrAlg.CanRun) THEN
  					StrAlg.isRuning := TRUE;
  					StrAlg.isEnded := FALSE;
  					StrAlg.hasError 	:= FALSE;

                                                    (*****************       OnRun       *****************)

  					cmd_for_Status := cmd;
  					source_for_Status := source;
  					command_error_for_Status := 0;
  				ELSE
  					StrAlg.isRuning := FALSE;
  					StrAlg.isEnded := FALSE;
  					StrAlg.hasError 	:= FALSE;

  					cmd_for_Status := 0;
  					source_for_Status := source;
  					command_error_for_Status := cmd;
  				END_IF;
  		(*cmdReset*) 2: 	StrAlg.isRuning := FALSE;
  				StrAlg.isEnded := FALSE;
  				StrAlg.hasError 	:= FALSE;
                                          (*****************       OnReset       *****************)

                                                    pompaj:= FALSE;
                                                    Kran6.inOpcCommandsDisabled:=FALSE;
  				cmd_for_Status := cmd;
  				source_for_Status := source;
  				command_error_for_Status := 0;
  	END_CASE;
  	resetCmdTimer(IN := false);
  	resetCmdTimerPriznak := TRUE;
  END_IF;
  lastCmd := cmd;

  resetCmdTimer(IN := resetCmdTimerPriznak, PT := T#5S);
  IF resetCmdTimer.Q THEN
  	resetCmdTimerPriznak := FALSE;
  	source_for_Status := 0;
  	cmd_for_Status := 0;
  	command_error_for_Status := 0;
  END_IF;

  StrAlg.status :=  SHL(BYTE_TO_DWORD(source_for_Status), 29)
  			OR SHL(BYTE_TO_DWORD(cmd_for_Status), 26)
  			OR SHL(BYTE_TO_DWORD(command_error_for_Status), 23)
  			OR SHL(BOOL_TO_DWORD(StrAlg.OpcCommandsDisabled ), 21)
  			OR SHL(BOOL_TO_DWORD(StrAlg.hasError),4)
  			OR SHL(BOOL_TO_DWORD(StrAlg.CanRun),2)
  			OR SHL(BOOL_TO_DWORD(StrAlg.isEnded),1)
  			OR BOOL_TO_DWORD(StrAlg.isRuning);
END_FUNCTION_BLOCK

FUNCTION_BLOCK fb_ph_Kran
  VAR_IN_OUT
    im : struct_Kran;
    StrPh : struct_PhaseAlgoritm;
  END_VAR
  VAR_INPUT
    act : TYPE_DualStateImAction;
    PhaseNumber : UINT;
  END_VAR
  VAR
    CommandFault_Trig : R_TRIG;
    reset_Trig : R_TRIG;
    _statusDualInput : TYPE_statusDualInput;
  END_VAR

  IF StrPh.run AND NOT StrPh.start THEN
  	StrPh.start := TRUE;
  	StrPh.top := FALSE;
  	StrPh.error := FALSE;
            StrPh.run:=FALSE;

  	CASE act OF
  		(*DualStateImAction.on*)   _on: im.inOpcCommandsDisabled:=TRUE;
                                                      im.inCommand_Alg := 1; (*cmd_open*)
  		(*DualStateImAction.off*) _off: im.inOpcCommandsDisabled:=TRUE;
                                                      im.inCommand_Alg := 2; (*cmd_close*)
  	END_CASE;
  END_IF;

  IF StrPh.start AND NOT StrPh.top THEN
                      CommandFault_Trig(CLK := im.CommandFault);
                      IF CommandFault_Trig.Q THEN
  	          StrPh.error := TRUE;
                      END_IF;

  		CASE act OF
  		(*_DualStateImAction.on*)    _on: StrPh.top := im.onStatus = _statusDualInput.STATUS_ON;
  		(*_DualStateImAction.off*)  _off: StrPh.top := im.onStatus = _statusDualInput.STATUS_OFF;
  		END_CASE;

  END_IF;

  IF StrPh.top THEN
  StrPh.error := FALSE;
  END_IF;

  reset_Trig(CLK := StrPh.reset);
  IF reset_Trig.Q THEN
  	StrPh.start := FALSE;
  	StrPh.error := FALSE;
  	StrPh.top := FALSE;
            StrPh.run:=FALSE;
            StrPh.reset:=FALSE;
  END_IF;

  StrPh.startStatus := SHL(BOOL_TO_DWORD(StrPh.start), PhaseNumber);
  StrPh.errorStatus := SHL(BOOL_TO_DWORD(StrPh.error), PhaseNumber);
  StrPh.topStatus := SHL(BOOL_TO_DWORD(StrPh.top), PhaseNumber);
END_FUNCTION_BLOCK

FUNCTION_BLOCK fb_ph_SectionSwitch
  VAR_IN_OUT
    im : struct_SectionSwitch;
  END_VAR
  VAR_INPUT
    act : TYPE_DualStateImAction;
    PhaseNumber : UINT;
  END_VAR
  VAR_IN_OUT
    StrPh : struct_PhaseAlgoritm;
  END_VAR
  VAR
    CommandFault_Trig : R_TRIG;
    reset_Trig : R_TRIG;
    _statusDualInput : TYPE_statusDualInput;
  END_VAR

  IF StrPh.run AND NOT StrPh.start THEN
  	StrPh.start := TRUE;
  	StrPh.top := FALSE;
  	StrPh.error := FALSE;
            StrPh.run:=FALSE;

  	CASE act OF
  		(*DualStateImAction.on*)   _on : im.inOpcCommandsDisabled:=TRUE;
                                                       im.inCommand_Alg := 1; (*cmd_open*)
  		(*DualStateImAction.off*) _off : im.inOpcCommandsDisabled:=TRUE;
                                                       im.inCommand_Alg := 2; (*cmd_close*)
  	END_CASE;
  END_IF;

  IF StrPh.start AND NOT StrPh.top THEN
                      CommandFault_Trig(CLK := im.CommandFault);
                      IF CommandFault_Trig.Q THEN
  	          StrPh.error := TRUE;
                      END_IF;

  		CASE act OF
  		(*_DualStateImAction.on*)    _on: StrPh.top := im.onStatus = _statusDualInput.STATUS_ON;
  		(*_DualStateImAction.off*)  _off: StrPh.top := im.onStatus = _statusDualInput.STATUS_OFF;
  		END_CASE;

  END_IF;

  IF StrPh.top THEN
  StrPh.error := FALSE;
  END_IF;

  reset_Trig(CLK := StrPh.reset);
  IF reset_Trig.Q THEN
  	StrPh.start := FALSE;
  	StrPh.error := FALSE;
  	StrPh.top := FALSE;
            StrPh.run:=FALSE;
            StrPh.reset:=FALSE;
  END_IF;

  StrPh.startStatus := SHL(BOOL_TO_DWORD(StrPh.start), PhaseNumber);
  StrPh.errorStatus := SHL(BOOL_TO_DWORD(StrPh.error), PhaseNumber);
  StrPh.topStatus := SHL(BOOL_TO_DWORD(StrPh.top), PhaseNumber);
END_FUNCTION_BLOCK

FUNCTION runIfNotRunningSO : BOOL
  VAR_IN_OUT
    so : struct_singleOutput;
  END_VAR
  VAR CONSTANT
    cmdRun : WORD := 1;
  END_VAR

  IF NOT so.Q THEN
                      so.inOpcCommandsDisabled:=TRUE;
  		so.inCommand_Alg:=cmdRun;
  END_IF;
END_FUNCTION

FUNCTION resetIfRunningSO : BOOL
  VAR_IN_OUT
    so : struct_singleOutput;
  END_VAR
  VAR CONSTANT
    cmdReset : WORD := 2;
  END_VAR

  IF so.Q THEN
                      so.inOpcCommandsDisabled:=TRUE;
  		so.inCommand_Alg:=cmdReset;
  END_IF;
END_FUNCTION

FUNCTION impulseSO : BOOL
  VAR_IN_OUT
    so : struct_singleOutput;
  END_VAR
  VAR CONSTANT
    cmdImpulse : WORD := 3;
  END_VAR

  IF NOT so.Q THEN
                      so.inOpcCommandsDisabled:=TRUE;
  		so.inCommand_Alg:=cmdImpulse;
  END_IF;
END_FUNCTION

FUNCTION_BLOCK NOAlg
  VAR_IN_OUT
    StrAlg : struct_Alg;
  END_VAR
  VAR
    kran4Close : struct_PhaseAlgoritm;
    mvOff : struct_PhaseAlgoritm;
    pnsOn : struct_PhaseAlgoritm;
    kran3bOpen : struct_PhaseAlgoritm;
    kran1Close : struct_PhaseAlgoritm;
    kran2Close : struct_PhaseAlgoritm;
    kran5Open : struct_PhaseAlgoritm;
    autoNuOff : struct_PhaseAlgoritm;
    autoPnsOff : struct_PhaseAlgoritm;
    pInNagLess100 : struct_PhaseAlgoritm;
    autoAvomOff : struct_PhaseAlgoritm;
    avom1cmdOff : struct_PhaseAlgoritm;
    avom2cmdOff : struct_PhaseAlgoritm;
    nu1off : struct_PhaseAlgoritm;
    nu2off : struct_PhaseAlgoritm;
    LowOil : struct_PhaseAlgoritm;
    waitCloseKran : struct_PhaseAlgoritm;
    pnsWaitOff : struct_PhaseAlgoritm;
    runUnsuccessful : struct_PhaseAlgoritm;
    fb_kran4Close : fb_ph_Kran;
    fb_mvOff : fb_ph_SectionSwitch;
    fb_pnsOn : fb_ph_Switch;
    fb_kran3bOpen : fb_ph_Kran;
    fb_kran1Close : fb_ph_Kran;
    fb_kran2Close : fb_ph_Kran;
    fb_kran5Open : fb_ph_Kran;
    fb_autoNuOff : fb_ph_algoritm;
    fb_autoPnsOff : fb_ph_algoritm;
    fb_pInNagLess100 : fb_ph_CustomPhase;
    fb_autoAvomOff : fb_ph_algoritm;
    fb_avom1cmdOff : fb_ph_Switch;
    fb_avom2cmdOff : fb_ph_Switch;
    fb_nu1off : fb_ph_OilPump;
    fb_nu2off : fb_ph_OilPump;
    fb_LowOil : fb_ph_WaitAnalogValue;
    fb_waitCloseKran : fb_ph_Timer;
    fb_pnsWaitOff : fb_ph_algoritm;
    fb_runUnsuccessful : fb_ph_CustomPhase;
    _sunpackerCommand : fb_sunpackerCommand;
    _statusAi : TYPE_StatusAi;
    _Answers : TYPE_Answers;
    _statusDualInput : TYPE_statusDualInput;
    _commandDualInput : TYPE_commandDualInput;
    _DualStateImAction : TYPE_DualStateImAction;
    _PhaseAlgoritmAction : TYPE_PhaseAlgoritmAction;
    source : BYTE;
    cmd : BYTE;
    lastCmd : BYTE;
    source_for_Status : BYTE;
    cmd_for_Status : BYTE;
    command_error_for_Status : BYTE;
    resetCmdTimer : TON;
    resetCmdTimerPriznak : BOOL;
  END_VAR
  VAR CONSTANT
    Ust_Pgaza : LREAL := 0.3;
  END_VAR
  VAR
    onInit : BOOL;
    waitReset : TON;
  END_VAR
  VAR_EXTERNAL
    IM : ImConfig;
    algoritms : AlgoritmsConfig;
    ai : AiConfig;
    protections : ProtectionsConfig;
    ModeGpa : TYPE_ModeGpa;
    algManager : struct_AlgoritmsManager;
    AlgTimers : struct_AlgTimers;
  END_VAR

  IF NOT onInit THEN

         fb_kran4Close(phaseNumber:=1, act:=_off);
              fb_mvOff(phaseNumber:=2, act:=_off);
              fb_pnsOn(phaseNumber:=3, act:=_on);
         fb_kran3bOpen(phaseNumber:=4, act:=_on);
         fb_kran1Close(phaseNumber:=5, act:=_off);
         fb_kran2Close(phaseNumber:=6, act:=_off);
          fb_kran5Open(phaseNumber:=7, act:=_on);
          fb_autoNuOff(phaseNumber:=8, act:=_reset, waitCompletion:=FALSE);
         fb_autoPnsOff(phaseNumber:=9, act:=_reset, waitCompletion:=FALSE);
      fb_pInNagLess100(phaseNumber:=10);
        fb_autoAvomOff(phaseNumber:=11, act:=_reset, waitCompletion:=FALSE);
        fb_avom1cmdOff(phaseNumber:=12, act:=_off);
        fb_avom2cmdOff(phaseNumber:=13, act:=_off);
             fb_nu1off(phaseNumber:=14, act:=_off);
             fb_nu2off(phaseNumber:=15, act:=_off);
      fb_waitCloseKran(phaseNumber:=16, delay:=T#240S);
             fb_LowOil(phaseNumber:=17);
         fb_pnsWaitOff(phaseNumber:=18, act:=_run, waitCompletion:=TRUE);
    fb_runUnsuccessful(phaseNumber:=20);

  onInit:=TRUE;
  END_IF;

         fb_kran4Close(StrPh:=kran4Close, Im:=Im.kran4);
              fb_mvOff(StrPh:=mvOff, Im:=Im.mv);
              fb_pnsOn(StrPh:=pnsOn, Im:=Im.pns);
         fb_kran3bOpen(StrPh:=kran3bOpen, Im:=Im.kran3b);
         fb_kran1Close(StrPh:=kran1Close, Im:=Im.kran1);
         fb_kran2Close(StrPh:=kran2Close, Im:=Im.kran2);
          fb_kran5Open(StrPh:=kran5Open, Im:=Im.kran5);
          fb_autoNuOff(StrPh:=autoNuOff, alg:=algoritms.autoNu);
         fb_autoPnsOff(StrPh:=autoPnsOff, alg:=algoritms.autoPns);
      fb_pInNagLess100(StrPh:=pInNagLess100);
        fb_autoAvomOff(StrPh:=autoAvomOff, alg:=algoritms.AutoAvom);
        fb_avom1cmdOff(StrPh:=avom1cmdOff, Im:=Im.v1_Avom);
        fb_avom2cmdOff(StrPh:=avom2cmdOff, Im:=Im.v2_Avom);
             fb_nu1off(StrPh:=nu1off, Im:=Im.nu1);
             fb_nu2off(StrPh:=nu2off, Im:=Im.nu2);
      fb_waitCloseKran(StrPh:=waitCloseKran, timer:=AlgTimers.NO_waitCloseKran);
             fb_LowOil(StrPh:=LowOil, ai:=ai.P_masla_smazki_nizkoe, less:=im.AutoPns_UstRun.value);
         fb_pnsWaitOff(StrPh:=pnsWaitOff, alg:=algoritms.vibegPNS, waitCompletion:=TRUE);
    fb_runUnsuccessful(StrPh:=runUnsuccessful);

  StrAlg.CanRun := StrAlg.inCanRun;
  StrAlg.OpcCommandsDisabled := StrAlg.inOpcCommandsDisabled;

  IF StrAlg.isRuning THEN

      StrAlg.hasError := kran4Close.error OR mvOff.error OR pnsOn.error OR kran3bOpen.error
      OR kran1Close.error OR kran2Close.error OR kran5Open.error OR runUnsuccessful.error;

      IF kran3bOpen.top THEN
          runPhase(kran1Close);
          runPhase(kran2Close);
      END_IF;

      IF kran4Close.top AND kran1Close.top AND kran2Close.top THEN
          runPhase(kran5Open);
      END_IF;

      IF kran5Open.top THEN
         resetDiProtection(protections.mvOff);
         runPhase(mvOff);
      END_IF;

      IF mvOff.top THEN
            runPhase(autoPnsOff);
  	runPhase(pInNagLess100);
  	runPhase(LowOil);
      END_IF;

      IF LowOil.start AND NOT LowOil.top THEN
         im.pns.inopcCommandsDisabled:=FALSE;
             IF (im.pns.onStatus = _statusDualInput.STATUS_ON) THEN
                 im.pns.inopcCommandsDisabled:=TRUE;
                 im.pns.inCommand_Alg:=BYTE_TO_WORD(_commandDualInput.CMD_OFF);
             END_IF;

      END_IF;

      IF autoPnsOff.top AND LowOil.top THEN
  	runPhase(pnsOn);
      END_IF;

     IF pInNagLess100.start AND NOT pInNagLess100.top THEN
  	pInNagLess100.top:=( ai.P_gaza_na_vkhode_nagnetatelia.interval >= _statusAi.NORMAL AND
            ai.P_gaza_na_vkhode_nagnetatelia.value < Ust_Pgaza ) AND
           (ai.P_gaza_na_vykhode_nagnetatelia.interval >= _statusAi.NORMAL AND
            ai.P_gaza_na_vykhode_nagnetatelia.value < Ust_Pgaza);

     END_IF;

     IF pInNagLess100.top THEN
     resetPhase(waitCloseKran);
     END_IF;

      IF pInNagLess100.top AND pnsOn.top THEN
  	ai.dPmaslo_gaz.Disabled_LA:=TRUE;
            ai.dPmaslo_gaz.Disabled_LW:=TRUE;
            IM.SingleSignals.dP_oilgaz_low.Disabled_Sig:=TRUE;
            resetAiProtection(protections.dP_maslogaz_LA);
            resetDiProtection(protections.dP_masloGaz_LowDI);

            runPhase(autoNuOff);
      END_IF;

      IF autoNuOff.top THEN
  	runPhase(nu1off);
            runPhase(nu2off);
      END_IF;

      IF nu1off.top AND  nu2off.top THEN
  	runPhase(pnsWaitOff);
      END_IF;

      IF waitCloseKran.top AND (NOT pInNagLess100.top) THEN
  	runUnsuccessful.error:=TRUE;
      END_IF;

      IF pnsWaitOff.top THEN
  	runPhase(autoAvomOff);
      END_IF;

      IF autoAvomOff.top THEN
  	runPhase(avom1cmdOff);
  	runPhase(avom2cmdOff);
      END_IF;

      IF avom1cmdOff.top AND avom2cmdOff.top THEN
  	waitReset(IN:=TRUE, PT:= T#2S);
      END_IF;

      IF waitReset.Q THEN
      resetIfRunning(algoritms.vibegPNS);
      algManager.nMode:=ModeGpa.MODE_STOP;
      resetIfRunning(StrAlg);
      END_IF;

      StrAlg.isEnded:= avom1cmdOff.top AND avom2cmdOff.top AND pnsWaitOff.top;
  END_IF;

  StrAlg.CanRun := StrAlg.inCanRun;
  StrAlg.OpcCommandsDisabled := StrAlg.inOpcCommandsDisabled;

  (* ---- Если управление с ВУ заблокировано, то  передаем команду из алгоритма ---- *)
  IF StrAlg.inOpcCommandsDisabled THEN
  	StrAlg.inCommand := StrAlg.inCommand_Alg;
  ELSE (* иначе передаем команду с АРМа*)
  	StrAlg.inCommand := StrAlg.inCommand_ARM;
  END_IF;

  _sunpackerCommand(command := StrAlg.inCommand);
  	source := _sunpackerCommand.source;
  	cmd := _sunpackerCommand.cmd;

  IF cmd <> 0 AND lastCmd <> cmd AND (((NOT StrAlg.opcCommandsDisabled) AND source > 0) OR source = 0) then
  	CASE BYTE_TO_INT(cmd) OF
  		(*cmdRun*) 1: 	IF (StrAlg.CanRun) THEN
  					StrAlg.isRuning := TRUE;
  					StrAlg.isEnded := FALSE;
  					StrAlg.hasError := FALSE;
  					(*****************       OnRun       *****************)

                                                    algManager.nMode:=ModeGpa.MODE_NO;
                                                    runIfNotRunningSO(IM.SingleOutputs.Lampa_NO);

                                                    runPhase(kran3bOpen);
                                                    runPhase(kran4Close);
                                                    runPhase(waitCloseKran);
                                                    runPhase(runUnsuccessful);

                                                    resetAiProtection(protections.Vibratciia_rotora_nagnetatelia_t1_HA);
                                                    resetAiProtection(protections.Vibratciia_rotora_nagnetatelia_t2_HA);
                                                    resetAiProtection(protections.Vibratciia_rotora_nagnetatelia_t3_HA);
                                                    resetAiProtection(protections.Vibratciia_rotora_nagnetatelia_t4_HA);
                                                    resetAiProtection(protections.Vibratciia_STD_t1_HA);
                                                    resetAiProtection(protections.Vibratciia_STD_t2_HA);
                                                    resetDiProtection(protections.Kran1sdvig);
                                                    resetDiProtection(protections.Kran2sdvig);

  					cmd_for_Status := cmd;
  					source_for_Status := source;
  					command_error_for_Status := 0;
  				ELSE
  					StrAlg.isRuning := FALSE;
  					StrAlg.isEnded := FALSE;
  					StrAlg.hasError 	:= FALSE;

  					cmd_for_Status := 0;
  					source_for_Status := source;
  					command_error_for_Status := cmd;
  				END_IF;
  		(*cmdReset*) 2: 	StrAlg.isRuning := FALSE;
  				StrAlg.isEnded := FALSE;
  				StrAlg.hasError 	:= FALSE;

                                           (*****************       OnReset       *****************)
                                          waitReset(IN:=FALSE);
                                          resetIfRunningSO(IM.SingleOutputs.Lampa_NO);
                                          resetIfRunning(algoritms.vibegPNS);
                                          impulseSO(Im.SingleOutputs.SbrosBREO);

                                          resetPhase(kran4Close);
                                          resetPhase(mvOff);
                                          resetPhase(pnsOn);
                                          resetPhase(kran3bOpen);
                                          resetPhase(kran1Close);
                                          resetPhase(kran2Close);
                                          resetPhase(kran5Open);
                                          resetPhase(autoNuOff);
                                          resetPhase(autoPnsOff);
                                          resetPhase(pInNagLess100);
  	                              resetPhase(autoAvomOff);
                                          resetPhase(avom1cmdOff);
                                          resetPhase(avom2cmdOff);
                                          resetPhase(nu1off);
                                          resetPhase(nu2off);
                                          resetPhase(LowOil);
                                          resetPhase(waitCloseKran);
                                          resetPhase(pnsWaitOff);
                                          resetPhase(runUnsuccessful);

  				cmd_for_Status := cmd;
  				source_for_Status := source;
  				command_error_for_Status := 0;
  	END_CASE;
  	resetCmdTimer(IN := false);
  	resetCmdTimerPriznak := TRUE;
  END_IF;
  lastCmd := cmd;

  resetCmdTimer(IN := resetCmdTimerPriznak, PT := T#5S);
  IF resetCmdTimer.Q THEN
  	resetCmdTimerPriznak := FALSE;
  	source_for_Status := 0;
  	cmd_for_Status := 0;
  	command_error_for_Status := 0;
  END_IF;

  StrAlg.Start:= kran4Close.startStatus
              OR mvOff.startStatus
              OR pnsOn.startStatus
              OR kran3bOpen.startStatus
              OR kran1Close.startStatus
              OR kran2Close.startStatus
              OR kran5Open.startStatus
              OR autoNuOff.startStatus
              OR autoPnsOff.startStatus
              OR pInNagLess100.startStatus
              OR autoAvomOff.startStatus
              OR avom1cmdOff.startStatus
              OR avom2cmdOff.startStatus
              OR nu1off.startStatus
              OR nu2off.startStatus
              OR LowOil.startStatus
              OR waitCloseKran.startStatus
              OR pnsWaitOff.startStatus
              OR runUnsuccessful.startStatus;

  StrAlg.Error:= kran4Close.errorStatus
              OR mvOff.errorStatus
              OR pnsOn.errorStatus
              OR kran3bOpen.errorStatus
              OR kran1Close.errorStatus
              OR kran2Close.errorStatus
              OR kran5Open.errorStatus
              OR autoNuOff.errorStatus
              OR autoPnsOff.errorStatus
              OR pInNagLess100.errorStatus
              OR autoAvomOff.errorStatus
              OR avom1cmdOff.errorStatus
              OR avom2cmdOff.errorStatus
              OR nu1off.errorStatus
              OR nu2off.errorStatus
              OR LowOil.errorStatus
              OR waitCloseKran.errorStatus
              OR pnsWaitOff.errorStatus
              OR runUnsuccessful.errorStatus;

  StrAlg.Top:=   kran4Close.topStatus
              OR mvOff.topStatus
              OR pnsOn.topStatus
              OR kran3bOpen.topStatus
              OR kran1Close.topStatus
              OR kran2Close.topStatus
              OR kran5Open.topStatus
              OR autoNuOff.topStatus
              OR autoPnsOff.topStatus
              OR pInNagLess100.topStatus
              OR autoAvomOff.topStatus
              OR avom1cmdOff.topStatus
              OR avom2cmdOff.topStatus
              OR nu1off.topStatus
              OR nu2off.topStatus
              OR LowOil.topStatus
              OR waitCloseKran.topStatus
              OR pnsWaitOff.topStatus
              OR runUnsuccessful.topStatus;

  (*TODO: TYPE PROGRAM CODE HERE*)
  StrAlg.status :=  SHL(BYTE_TO_DWORD(source_for_Status), 29)
  			OR SHL(BYTE_TO_DWORD(cmd_for_Status), 26)
  			OR SHL(BYTE_TO_DWORD(command_error_for_Status), 23)
  			OR SHL(BOOL_TO_DWORD(StrAlg.OpcCommandsDisabled ), 21)
  			OR SHL(BOOL_TO_DWORD(StrAlg.hasError),4)
  			OR SHL(BOOL_TO_DWORD(StrAlg.CanRun),2)
  			OR SHL(BOOL_TO_DWORD(StrAlg.isEnded),1)
  			OR BOOL_TO_DWORD(StrAlg.isRuning);
END_FUNCTION_BLOCK

FUNCTION stopPusk : BOOL
  VAR_IN_OUT
    algoritms : AlgoritmsConfig;
  END_VAR

  resetAndDisable(alg:=algoritms.Apusk);
  resetAndDisable(alg:=algoritms.SemiAutoPusk);
  resetAndDisable(alg:=algoritms.testPms);
  resetAndDisable(alg:=algoritms.puskV);
  resetAndDisable(alg:=algoritms.puskK);
  resetAndDisable(alg:=algoritms.testdPmg);
  resetAndDisable(alg:=algoritms.ppu);
  resetAndDisable(alg:=algoritms.puskOilSystem);
  resetAndDisable(alg:=algoritms.filling);
  resetAndDisable(alg:=algoritms.engineRun);
  resetAndDisable(alg:=algoritms.RingToLine);
  resetAndDisable(alg:=algoritms.LineToRing);
END_FUNCTION

FUNCTION_BLOCK AOAlg
  VAR_IN_OUT
    StrAlg : struct_Alg;
  END_VAR
  VAR
    kran4Close : struct_PhaseAlgoritm;
    mvOff : struct_PhaseAlgoritm;
    pnsOn : struct_PhaseAlgoritm;
    kran3bOpen : struct_PhaseAlgoritm;
    kran1Close : struct_PhaseAlgoritm;
    kran2Close : struct_PhaseAlgoritm;
    kran5Open : struct_PhaseAlgoritm;
    autoNuOff : struct_PhaseAlgoritm;
    autoPnsOff : struct_PhaseAlgoritm;
    pInNagLess100 : struct_PhaseAlgoritm;
    autoAvomOff : struct_PhaseAlgoritm;
    avom1cmdOff : struct_PhaseAlgoritm;
    avom2cmdOff : struct_PhaseAlgoritm;
    nu1off : struct_PhaseAlgoritm;
    nu2off : struct_PhaseAlgoritm;
    LowOil : struct_PhaseAlgoritm;
    waitKran : struct_PhaseAlgoritm;
    pnsWaitOff : struct_PhaseAlgoritm;
    runUnsuccessful : struct_PhaseAlgoritm;
    fb_kran4Close : fb_ph_Kran;
    fb_mvOff : fb_ph_SectionSwitch;
    fb_pnsOn : fb_ph_Switch;
    fb_kran3bOpen : fb_ph_Kran;
    fb_kran1Close : fb_ph_Kran;
    fb_kran2Close : fb_ph_Kran;
    fb_kran5Open : fb_ph_Kran;
    fb_autoNuOff : fb_ph_algoritm;
    fb_autoPnsOff : fb_ph_algoritm;
    fb_pInNagLess100 : fb_ph_CustomPhase;
    fb_autoAvomOff : fb_ph_algoritm;
    fb_avom1cmdOff : fb_ph_Switch;
    fb_avom2cmdOff : fb_ph_Switch;
    fb_nu1off : fb_ph_OilPump;
    fb_nu2off : fb_ph_OilPump;
    fb_LowOil : fb_ph_WaitAnalogValue;
    fb_waitKran : fb_ph_Timer;
    fb_pnsWaitOff : fb_ph_algoritm;
    fb_runUnsuccessful : fb_ph_CustomPhase;
    _sunpackerCommand : fb_sunpackerCommand;
    _statusAi : TYPE_StatusAi;
    _Answers : TYPE_Answers;
    _statusDualInput : TYPE_statusDualInput;
    _commandDualInput : TYPE_commandDualInput;
    _DualStateImAction : TYPE_DualStateImAction;
    _PhaseAlgoritmAction : TYPE_PhaseAlgoritmAction;
    source : BYTE;
    cmd : BYTE;
    lastCmd : BYTE;
    source_for_Status : BYTE;
    cmd_for_Status : BYTE;
    command_error_for_Status : BYTE;
    resetCmdTimer : TON;
    resetCmdTimerPriznak : BOOL;
  END_VAR
  VAR CONSTANT
    Ust_Pgaza : LREAL := 0.3;
  END_VAR
  VAR
    onInit : BOOL;
    waitReset : TON;
  END_VAR
  VAR_EXTERNAL
    IM : ImConfig;
    algoritms : AlgoritmsConfig;
    ai : AiConfig;
    protections : ProtectionsConfig;
    ModeGpa : TYPE_ModeGpa;
    algManager : struct_AlgoritmsManager;
    AlgTimers : struct_AlgTimers;
    PMcommand : TYPE_CommandsPotectionsManager;
    protectManager : struct_ProtectionsManager;
  END_VAR
